LIN {X 0,Y 453.492,Z 301.489,A -85,B 0,C 180,E1 -8435.264,E2 -8435.264} C_VEL
LIN {X 0,Y 453.473,Z 301.492,A -85,B 0,C 180,E1 -8438.414,E2 -8438.414} C_VEL
LIN {X 0,Y 453.514,Z 301.48,A -85,B 0,C 180,E1 -8441.008,E2 -8441.008} C_VEL
LIN {X 0,Y 453.56,Z 301.483,A -85,B 0,C 180,E1 -8443.879,E2 -8443.879} C_VEL
LIN {X 0,Y 453.555,Z 301.485,A -85,B 0,C 180,E1 -8447.47,E2 -8447.47} C_VEL
LIN {X 0,Y 453.584,Z 301.465,A -85,B 0,C 180,E1 -8451.086,E2 -8451.086} C_VEL
LIN {X 0,Y 453.668,Z 301.472,A -85,B 0,C 180,E1 -8453.774,E2 -8453.774} C_VEL
LIN {X 0,Y 453.755,Z 301.46,A -85,B 0,C 180,E1 -8457.336,E2 -8457.336} C_VEL
LIN {X 0,Y 453.812,Z 301.433,A -85,B 0,C 180,E1 -8460,E2 -8460} C_VEL
LIN {X 0,Y 453.735,Z 301.456,A -85,B 0,C 180,E1 -8462.663,E2 -8462.663} C_VEL
LIN {X 0,Y 453.667,Z 301.47,A -85,B 0,C 180,E1 -8466.225,E2 -8466.225} C_VEL
LIN {X 0,Y 453.583,Z 301.473,A -85,B 0,C 180,E1 -8468.913,E2 -8468.913} C_VEL
LIN {X 0,Y 453.553,Z 301.48,A -85,B 0,C 180,E1 -8472.529,E2 -8472.529} C_VEL
LIN {X 0,Y 453.534,Z 301.486,A -85,B 0,C 180,E1 -8476.196,E2 -8476.196} C_VEL
LIN {X 0,Y 453.51,Z 301.48,A -85,B 0,C 180,E1 -8479.04,E2 -8479.04} C_VEL
LIN {X 0,Y 453.466,Z 301.493,A -85,B 0,C 180,E1 -8481.836,E2 -8481.836} C_VEL
LIN {X 0,Y 453.504,Z 301.496,A -85,B 0,C 180,E1 -8484.734,E2 -8484.734} C_VEL
LIN {X 0,Y 453.523,Z 301.478,A -85,B 0,C 180,E1 -8487.96,E2 -8487.96} C_VEL
LIN {X 0,Y 453.474,Z 301.501,A -85,B 0,C 180,E1 -8490.759,E2 -8490.759} C_VEL
LIN {X 0,Y 453.468,Z 301.489,A -85,B 0,C 180,E1 -8493.913,E2 -8493.913} C_VEL
LIN {X 0,Y 453.462,Z 301.499,A -85,B 0,C 180,E1 -8497.188,E2 -8497.188} C_VEL
LIN {X 0,Y 453.522,Z 301.486,A -85,B 0,C 180,E1 -8499.446,E2 -8499.446} C_VEL
LIN {X 0,Y 453.481,Z 301.498,A -85,B 0,C 180,E1 -8502.992,E2 -8502.992} C_VEL
LIN {X 0,Y 453.465,Z 301.49,A -85,B 0,C 180,E1 -8505.78,E2 -8505.78} C_VEL
LIN {X 0,Y 453.507,Z 301.481,A -85,B 0,C 180,E1 -8509.406,E2 -8509.406} C_VEL
LIN {X 0,Y 453.466,Z 301.501,A -85,B 0,C 180,E1 -8512.224,E2 -8512.224} C_VEL
LIN {X 0,Y 453.482,Z 301.478,A -85,B 0,C 180,E1 -8515.223,E2 -8515.223} C_VEL
LIN {X 0,Y 453.461,Z 301.502,A -85,B 0,C 180,E1 -8518.475,E2 -8518.475} C_VEL
LIN {X 0,Y 453.532,Z 301.487,A -85,B 0,C 180,E1 -8522.039,E2 -8522.039} C_VEL
LIN {X 0,Y 453.509,Z 301.493,A -85,B 0,C 180,E1 -8525.266,E2 -8525.266} C_VEL
LIN {X 0,Y 453.475,Z 301.501,A -85,B 0,C 180,E1 -8528.415,E2 -8528.415} C_VEL
LIN {X 0,Y 453.517,Z 301.493,A -85,B 0,C 180,E1 -8531.009,E2 -8531.009} C_VEL
LIN {X 0,Y 453.564,Z 301.49,A -85,B 0,C 180,E1 -8533.88,E2 -8533.88} C_VEL
LIN {X 0,Y 453.559,Z 301.488,A -85,B 0,C 180,E1 -8537.471,E2 -8537.471} C_VEL
LIN {X 0,Y 453.589,Z 301.484,A -85,B 0,C 180,E1 -8541.087,E2 -8541.087} C_VEL
LIN {X 0,Y 453.634,Z 301.478,A -85,B 0,C 180,E1 -8543.101,E2 -8543.101} C_VEL
LIN {X 0,Y 452.949,Z 301.567,A -85,B 0,C 180,E1 -8543.841,E2 -8543.841} C_VEL
LIN {X 0,Y 450.001,Z 301.932,A -85,B 0,C 180,E1 -8545.043,E2 -8545.043} C_VEL
LIN {X 0,Y 447.578,Z 302.236,A -85,B 0,C 180,E1 -8546.012,E2 -8546.012} C_VEL
LIN {X 0,Y 446.643,Z 302.351,A -85,B 0,C 180,E1 -8546.763,E2 -8546.763} C_VEL
LIN {X 0,Y 446.623,Z 302.352,A -85,B 0,C 180,E1 -8547.016,E2 -8547.016} C_VEL
LIN {X 0,Y 446.791,Z 302.334,A -85,B 0,C 180,E1 -8550,E2 -8550} C_VEL
LIN {X 0,Y 446.706,Z 302.342,A -85,B 0,C 180,E1 -8552.705,E2 -8552.705} C_VEL
LIN {X 0,Y 446.644,Z 302.351,A -85,B 0,C 180,E1 -8556.324,E2 -8556.324} C_VEL
LIN {X 0,Y 446.534,Z 302.364,A -85,B 0,C 180,E1 -8559.055,E2 -8559.055} C_VEL
LIN {X 0,Y 446.517,Z 302.365,A -85,B 0,C 180,E1 -8562.73,E2 -8562.73} C_VEL
LIN {X 0,Y 446.492,Z 302.37,A -85,B 0,C 180,E1 -8566.228,E2 -8566.228} C_VEL
LIN {X 0,Y 446.465,Z 302.373,A -85,B 0,C 180,E1 -8569.303,E2 -8569.303} C_VEL
LIN {X 0,Y 446.414,Z 302.379,A -85,B 0,C 180,E1 -8572.199,E2 -8572.199} C_VEL
LIN {X 0,Y 446.453,Z 302.374,A -85,B 0,C 180,E1 -8575.152,E2 -8575.152} C_VEL
LIN {X 0,Y 446.479,Z 302.363,A -85,B 0,C 180,E1 -8578.178,E2 -8578.178} C_VEL
LIN {X 0,Y 446.414,Z 302.379,A -85,B 0,C 180,E1 -8581.775,E2 -8581.775} C_VEL
LIN {X 0,Y 446.423,Z 302.356,A -85,B 0,C 180,E1 -8584.523,E2 -8584.523} C_VEL
LIN {X 0,Y 446.425,Z 302.375,A -85,B 0,C 180,E1 -8588.082,E2 -8588.082} C_VEL
LIN {X 0,Y 446.435,Z 302.358,A -85,B 0,C 180,E1 -8590.92,E2 -8590.92} C_VEL
LIN {X 0,Y 446.414,Z 302.367,A -85,B 0,C 180,E1 -8593.843,E2 -8593.843} C_VEL
LIN {X 0,Y 446.436,Z 302.372,A -85,B 0,C 180,E1 -8596.397,E2 -8596.397} C_VEL
LIN {X 0,Y 446.46,Z 302.367,A -85,B 0,C 180,E1 -8599.805,E2 -8599.805} C_VEL
LIN {X 0,Y 446.424,Z 302.374,A -85,B 0,C 180,E1 -8602.123,E2 -8602.123} C_VEL
LIN {X 0,Y 446.421,Z 302.368,A -85,B 0,C 180,E1 -8605.477,E2 -8605.477} C_VEL
LIN {X 0,Y 446.41,Z 302.377,A -85,B 0,C 180,E1 -8608.7,E2 -8608.7} C_VEL
LIN {X 0,Y 446.475,Z 302.356,A -85,B 0,C 180,E1 -8611.821,E2 -8611.821} C_VEL
LIN {X 0,Y 446.447,Z 302.369,A -85,B 0,C 180,E1 -8614.848,E2 -8614.848} C_VEL
LIN {X 0,Y 446.438,Z 302.369,A -85,B 0,C 180,E1 -8618.245,E2 -8618.245} C_VEL
LIN {X 0,Y 446.447,Z 302.361,A -85,B 0,C 180,E1 -8621.649,E2 -8621.649} C_VEL
LIN {X 0,Y 446.498,Z 302.364,A -85,B 0,C 180,E1 -8624.48,E2 -8624.48} C_VEL
LIN {X 0,Y 446.506,Z 302.359,A -85,B 0,C 180,E1 -8627.384,E2 -8627.384} C_VEL
LIN {X 0,Y 446.528,Z 302.348,A -85,B 0,C 180,E1 -8630.945,E2 -8630.945} C_VEL
LIN {X 0,Y 446.636,Z 302.346,A -85,B 0,C 180,E1 -8633.677,E2 -8633.677} C_VEL
LIN {X 0,Y 446.682,Z 302.335,A -85,B 0,C 180,E1 -8637.295,E2 -8637.295} C_VEL
LIN {X 0,Y 446.783,Z 302.308,A -85,B 0,C 180,E1 -8640.001,E2 -8640.001} C_VEL
LIN {X 0,Y 446.699,Z 302.339,A -85,B 0,C 180,E1 -8642.706,E2 -8642.706} C_VEL
LIN {X 0,Y 446.637,Z 302.348,A -85,B 0,C 180,E1 -8646.324,E2 -8646.324} C_VEL
LIN {X 0,Y 446.53,Z 302.342,A -85,B 0,C 180,E1 -8649.056,E2 -8649.056} C_VEL
LIN {X 0,Y 446.513,Z 302.365,A -85,B 0,C 180,E1 -8652.73,E2 -8652.73} C_VEL
LIN {X 0,Y 446.488,Z 302.365,A -85,B 0,C 180,E1 -8656.229,E2 -8656.229} C_VEL
LIN {X 0,Y 446.462,Z 302.356,A -85,B 0,C 180,E1 -8659.304,E2 -8659.304} C_VEL
LIN {X 0,Y 446.41,Z 302.376,A -85,B 0,C 180,E1 -8662.2,E2 -8662.2} C_VEL
LIN {X 0,Y 446.436,Z 302.364,A -85,B 0,C 180,E1 -8665.154,E2 -8665.154} C_VEL
LIN {X 0,Y 446.479,Z 302.36,A -85,B 0,C 180,E1 -8668.18,E2 -8668.18} C_VEL
LIN {X 0,Y 446.408,Z 302.374,A -85,B 0,C 180,E1 -8671.301,E2 -8671.301} C_VEL
LIN {X 0,Y 446.416,Z 302.37,A -85,B 0,C 180,E1 -8674.525,E2 -8674.525} C_VEL
LIN {X 0,Y 446.408,Z 302.381,A -85,B 0,C 180,E1 -8678.08,E2 -8678.08} C_VEL
LIN {X 0,Y 446.422,Z 302.372,A -85,B 0,C 180,E1 -8680.918,E2 -8680.918} C_VEL
LIN {X 0,Y 446.395,Z 302.38,A -85,B 0,C 180,E1 -8683.847,E2 -8683.847} C_VEL
LIN {X 0,Y 446.396,Z 302.381,A -85,B 0,C 180,E1 -8686.404,E2 -8686.404} C_VEL
LIN {X 0,Y 446.419,Z 302.361,A -85,B 0,C 180,E1 -8689.084,E2 -8689.084} C_VEL
LIN {X 0,Y 446.403,Z 302.382,A -85,B 0,C 180,E1 -8692.122,E2 -8692.122} C_VEL
LIN {X 0,Y 446.427,Z 302.373,A -85,B 0,C 180,E1 -8695.478,E2 -8695.478} C_VEL
LIN {X 0,Y 446.416,Z 302.38,A -85,B 0,C 180,E1 -8698.7,E2 -8698.7} C_VEL
LIN {X 0,Y 446.523,Z 302.561,A -85,B 0,C 180,E1 -8701.813,E2 -8701.813} C_VEL
LIN {X 0,Y 448.386,Z 312.725,A -85,B 0,C 180,E1 -8704.467,E2 -8704.467} C_VEL
LIN {X 0,Y 448.438,Z 317.528,A -85,B 0,C 180,E1 -8705.649,E2 -8705.649} C_VEL
LIN {X 0,Y 447.685,Z 331.236,A -85,B 0,C 180,E1 -8708.835,E2 -8708.835} C_VEL
LIN {X 0,Y 447.04,Z 343.412,A -85,B 0,C 180,E1 -8711.674,E2 -8711.674} C_VEL
LIN {X 0,Y 446.989,Z 345.405,A -85,B 0,C 180,E1 -8712.117,E2 -8712.117} C_VEL
LIN {X 0,Y 447.514,Z 348.844,A -85,B 0,C 180,E1 -8712.245,E2 -8712.245} C_VEL
LIN {X 0,Y 450.815,Z 368.098,A -85,B 0,C 180,E1 -8712.692,E2 -8712.692} C_VEL
LIN {X 0,Y 450.115,Z 450.358,A -85,B 0,C 180,E1 -8714.027,E2 -8714.027} C_VEL
LIN {X 0,Y 449.794,Z 461.123,A -85,B 0,C 180,E1 -8714.306,E2 -8714.306} C_VEL
LIN {X 0,Y 449.474,Z 470.223,A -85,B 0,C 180,E1 -8714.643,E2 -8714.643} C_VEL
LIN {X 0,Y 448.987,Z 480.584,A -85,B 0,C 180,E1 -8715.149,E2 -8715.149} C_VEL
LIN {X 0,Y 448.533,Z 489.719,A -85,B 0,C 180,E1 -8715.713,E2 -8715.713} C_VEL
LIN {X 0,Y 448.044,Z 498.716,A -85,B 0,C 180,E1 -8716.392,E2 -8716.392} C_VEL
LIN {X 0,Y 447.604,Z 507.306,A -85,B 0,C 180,E1 -8717.172,E2 -8717.172} C_VEL
LIN {X 0,Y 447.186,Z 514.844,A -85,B 0,C 180,E1 -8717.981,E2 -8717.981} C_VEL
LIN {X 0,Y 446.7,Z 522.063,A -85,B 0,C 180,E1 -8718.888,E2 -8718.888} C_VEL
LIN {X 0,Y 446.377,Z 528.266,A -85,B 0,C 180,E1 -8719.798,E2 -8719.798} C_VEL
LIN {X 0,Y 446.006,Z 534.803,A -85,B 0,C 180,E1 -8720.934,E2 -8720.934} C_VEL
LIN {X 0,Y 445.838,Z 539.306,A -85,B 0,C 180,E1 -8721.844,E2 -8721.844} C_VEL
LIN {X 0,Y 445.581,Z 544.797,A -85,B 0,C 180,E1 -8723.207,E2 -8723.207} C_VEL
LIN {X 0,Y 445.479,Z 549.118,A -85,B 0,C 180,E1 -8724.569,E2 -8724.569} C_VEL
LIN {X 0,Y 445.414,Z 551.482,A -85,B 0,C 180,E1 -8725.475,E2 -8725.475} C_VEL
LIN {X 0,Y 445.433,Z 554.666,A -85,B 0,C 180,E1 -8727.287,E2 -8727.287} C_VEL
LIN {X 0,Y 445.356,Z 555.721,A -85,B 0,C 180,E1 -8728.191,E2 -8728.191} C_VEL
LIN {X 0,Y 445.339,Z 556.308,A -85,B 0,C 180,E1 -8729.096,E2 -8729.096} C_VEL
LIN {X 0,Y 445.339,Z 556.308,A -85,B 0,C 180,E1 -8730.904,E2 -8730.904} C_VEL
LIN {X 0,Y 445.356,Z 555.721,A -85,B 0,C 180,E1 -8731.809,E2 -8731.809} C_VEL
LIN {X 0,Y 445.433,Z 554.666,A -85,B 0,C 180,E1 -8732.713,E2 -8732.713} C_VEL
LIN {X 0,Y 445.414,Z 551.482,A -85,B 0,C 180,E1 -8734.525,E2 -8734.525} C_VEL
LIN {X 0,Y 445.471,Z 547.36,A -85,B 0,C 180,E1 -8736.044,E2 -8736.044} C_VEL
LIN {X 0,Y 445.637,Z 543.135,A -85,B 0,C 180,E1 -8737.248,E2 -8737.248} C_VEL
LIN {X 0,Y 445.897,Z 537.114,A -85,B 0,C 180,E1 -8738.611,E2 -8738.611} C_VEL
LIN {X 0,Y 446.217,Z 531.018,A -85,B 0,C 180,E1 -8739.748,E2 -8739.748} C_VEL
LIN {X 0,Y 446.506,Z 525.317,A -85,B 0,C 180,E1 -8740.658,E2 -8740.658} C_VEL
LIN {X 0,Y 447.064,Z 516.763,A -85,B 0,C 180,E1 -8741.792,E2 -8741.792} C_VEL
LIN {X 0,Y 447.541,Z 508.582,A -85,B 0,C 180,E1 -8742.7,E2 -8742.7} C_VEL
LIN {X 0,Y 447.964,Z 500.142,A -85,B 0,C 180,E1 -8743.489,E2 -8743.489} C_VEL
LIN {X 0,Y 448.474,Z 491.352,A -85,B 0,C 180,E1 -8744.173,E2 -8744.173} C_VEL
LIN {X 0,Y 448.961,Z 481.592,A -85,B 0,C 180,E1 -8744.794,E2 -8744.794} C_VEL
LIN {X 0,Y 449.367,Z 472.798,A -85,B 0,C 180,E1 -8745.244,E2 -8745.244} C_VEL
LIN {X 0,Y 449.75,Z 462.871,A -85,B 0,C 180,E1 -8745.637,E2 -8745.637} C_VEL
LIN {X 0,Y 450.049,Z 453.021,A -85,B 0,C 180,E1 -8745.917,E2 -8745.917} C_VEL
LIN {X 0,Y 450.317,Z 427.887,A -85,B 0,C 180,E1 -8746.353,E2 -8746.353} C_VEL
LIN {X 0,Y 450.703,Z 367.244,A -85,B 0,C 180,E1 -8747.326,E2 -8747.326} C_VEL
LIN {X 0,Y 447.009,Z 345.81,A -85,B 0,C 180,E1 -8747.844,E2 -8747.844} C_VEL
LIN {X 0,Y 447.009,Z 344.423,A -85,B 0,C 180,E1 -8748.076,E2 -8748.076} C_VEL
LIN {X 0,Y 447.714,Z 331.421,A -85,B 0,C 180,E1 -8751.164,E2 -8751.164} C_VEL
LIN {X 0,Y 448.576,Z 316.323,A -85,B 0,C 180,E1 -8754.672,E2 -8754.672} C_VEL
LIN {X 0,Y 448.193,Z 311.699,A -85,B 0,C 180,E1 -8755.794,E2 -8755.794} C_VEL
LIN {X 0,Y 446.51,Z 302.392,A -85,B 0,C 180,E1 -8758.259,E2 -8758.259} C_VEL
LIN {X 0,Y 446.419,Z 302.377,A -85,B 0,C 180,E1 -8761.774,E2 -8761.774} C_VEL
LIN {X 0,Y 446.427,Z 302.374,A -85,B 0,C 180,E1 -8764.522,E2 -8764.522} C_VEL
LIN {X 0,Y 446.409,Z 302.38,A -85,B 0,C 180,E1 -8768.078,E2 -8768.078} C_VEL
LIN {X 0,Y 446.416,Z 302.364,A -85,B 0,C 180,E1 -8771.391,E2 -8771.391} C_VEL
LIN {X 0,Y 446.447,Z 302.37,A -85,B 0,C 180,E1 -8775.103,E2 -8775.103} C_VEL
LIN {X 0,Y 446.424,Z 302.372,A -85,B 0,C 180,E1 -8778.608,E2 -8778.608} C_VEL
LIN {X 0,Y 446.433,Z 302.368,A -85,B 0,C 180,E1 -8780.971,E2 -8780.971} C_VEL
LIN {X 0,Y 446.412,Z 302.371,A -85,B 0,C 180,E1 -8784.373,E2 -8784.373} C_VEL
LIN {X 0,Y 446.41,Z 302.374,A -85,B 0,C 180,E1 -8787.637,E2 -8787.637} C_VEL
LIN {X 0,Y 446.442,Z 302.369,A -85,B 0,C 180,E1 -8790.79,E2 -8790.79} C_VEL
LIN {X 0,Y 446.471,Z 302.36,A -85,B 0,C 180,E1 -8793.848,E2 -8793.848} C_VEL
LIN {X 0,Y 446.418,Z 302.373,A -85,B 0,C 180,E1 -8796.822,E2 -8796.822} C_VEL
LIN {X 0,Y 446.437,Z 302.364,A -85,B 0,C 180,E1 -8799.736,E2 -8799.736} C_VEL
LIN {X 0,Y 446.455,Z 302.357,A -85,B 0,C 180,E1 -8802.596,E2 -8802.596} C_VEL
LIN {X 0,Y 446.464,Z 302.373,A -85,B 0,C 180,E1 -8805.412,E2 -8805.412} C_VEL
LIN {X 0,Y 446.51,Z 302.355,A -85,B 0,C 180,E1 -8808.192,E2 -8808.192} C_VEL
LIN {X 0,Y 446.591,Z 302.345,A -85,B 0,C 180,E1 -8811.857,E2 -8811.857} C_VEL
LIN {X 0,Y 446.636,Z 302.346,A -85,B 0,C 180,E1 -8814.582,E2 -8814.582} C_VEL
LIN {X 0,Y 446.699,Z 302.339,A -85,B 0,C 180,E1 -8817.294,E2 -8817.294} C_VEL
LIN {X 0,Y 446.783,Z 302.308,A -85,B 0,C 180,E1 -8819.999,E2 -8819.999} C_VEL
LIN {X 0,Y 446.683,Z 302.335,A -85,B 0,C 180,E1 -8822.705,E2 -8822.705} C_VEL
LIN {X 0,Y 446.636,Z 302.346,A -85,B 0,C 180,E1 -8826.323,E2 -8826.323} C_VEL
LIN {X 0,Y 446.528,Z 302.348,A -85,B 0,C 180,E1 -8829.055,E2 -8829.055} C_VEL
LIN {X 0,Y 446.514,Z 302.359,A -85,B 0,C 180,E1 -8832.729,E2 -8832.729} C_VEL
LIN {X 0,Y 446.486,Z 302.364,A -85,B 0,C 180,E1 -8836.228,E2 -8836.228} C_VEL
LIN {X 0,Y 446.459,Z 302.357,A -85,B 0,C 180,E1 -8839.303,E2 -8839.303} C_VEL
LIN {X 0,Y 446.408,Z 302.373,A -85,B 0,C 180,E1 -8842.2,E2 -8842.2} C_VEL
LIN {X 0,Y 446.447,Z 302.369,A -85,B 0,C 180,E1 -8845.152,E2 -8845.152} C_VEL
LIN {X 0,Y 446.475,Z 302.356,A -85,B 0,C 180,E1 -8848.179,E2 -8848.179} C_VEL
LIN {X 0,Y 446.41,Z 302.377,A -85,B 0,C 180,E1 -8851.3,E2 -8851.3} C_VEL
LIN {X 0,Y 446.421,Z 302.368,A -85,B 0,C 180,E1 -8854.523,E2 -8854.523} C_VEL
LIN {X 0,Y 446.428,Z 302.375,A -85,B 0,C 180,E1 -8858.083,E2 -8858.083} C_VEL
LIN {X 0,Y 446.436,Z 302.369,A -85,B 0,C 180,E1 -8860.921,E2 -8860.921} C_VEL
LIN {X 0,Y 446.434,Z 302.372,A -85,B 0,C 180,E1 -8863.841,E2 -8863.841} C_VEL
LIN {X 0,Y 446.412,Z 302.362,A -85,B 0,C 180,E1 -8866.401,E2 -8866.401} C_VEL
LIN {X 0,Y 446.458,Z 302.36,A -85,B 0,C 180,E1 -8869.805,E2 -8869.805} C_VEL
LIN {X 0,Y 446.421,Z 302.377,A -85,B 0,C 180,E1 -8872.124,E2 -8872.124} C_VEL
LIN {X 0,Y 446.423,Z 302.356,A -85,B 0,C 180,E1 -8875.477,E2 -8875.477} C_VEL
LIN {X 0,Y 446.41,Z 302.377,A -85,B 0,C 180,E1 -8878.7,E2 -8878.7} C_VEL
LIN {X 0,Y 446.479,Z 302.363,A -85,B 0,C 180,E1 -8881.822,E2 -8881.822} C_VEL
LIN {X 0,Y 446.453,Z 302.374,A -85,B 0,C 180,E1 -8884.848,E2 -8884.848} C_VEL
LIN {X 0,Y 446.443,Z 302.377,A -85,B 0,C 180,E1 -8888.245,E2 -8888.245} C_VEL
LIN {X 0,Y 446.453,Z 302.374,A -85,B 0,C 180,E1 -8891.649,E2 -8891.649} C_VEL
LIN {X 0,Y 446.503,Z 302.369,A -85,B 0,C 180,E1 -8894.48,E2 -8894.48} C_VEL
LIN {X 0,Y 446.514,Z 302.369,A -85,B 0,C 180,E1 -8898.193,E2 -8898.193} C_VEL
LIN {X 0,Y 446.596,Z 302.358,A -85,B 0,C 180,E1 -8901.858,E2 -8901.858} C_VEL
LIN {X 0,Y 446.643,Z 302.351,A -85,B 0,C 180,E1 -8904.583,E2 -8904.583} C_VEL
LIN {X 0,Y 446.623,Z 302.352,A -85,B 0,C 180,E1 -8907.016,E2 -8907.016} C_VEL
LIN {X 0,Y 446.106,Z 302.419,A -85,B 0,C 180,E1 -8907.769,E2 -8907.769} C_VEL
LIN {X 0,Y 443.288,Z 302.771,A -85,B 0,C 180,E1 -8908.992,E2 -8908.992} C_VEL
LIN {X 0,Y 440.801,Z 303.081,A -85,B 0,C 180,E1 -8909.979,E2 -8909.979} C_VEL
LIN {X 0,Y 439.712,Z 303.214,A -85,B 0,C 180,E1 -8910.742,E2 -8910.742} C_VEL
LIN {X 0,Y 439.618,Z 303.225,A -85,B 0,C 180,E1 -8911.001,E2 -8911.001} C_VEL
LIN {X 0,Y 439.653,Z 303.221,A -85,B 0,C 180,E1 -8912.749,E2 -8912.749} C_VEL
LIN {X 0,Y 439.615,Z 303.226,A -85,B 0,C 180,E1 -8916.425,E2 -8916.425} C_VEL
LIN {X 0,Y 439.496,Z 303.241,A -85,B 0,C 180,E1 -8919.201,E2 -8919.201} C_VEL
LIN {X 0,Y 439.461,Z 303.244,A -85,B 0,C 180,E1 -8922.937,E2 -8922.937} C_VEL
LIN {X 0,Y 439.443,Z 303.247,A -85,B 0,C 180,E1 -8926.349,E2 -8926.349} C_VEL
LIN {X 0,Y 439.398,Z 303.255,A -85,B 0,C 180,E1 -8929.626,E2 -8929.626} C_VEL
LIN {X 0,Y 439.361,Z 303.256,A -85,B 0,C 180,E1 -8932.575,E2 -8932.575} C_VEL
LIN {X 0,Y 439.401,Z 303.254,A -85,B 0,C 180,E1 -8935.584,E2 -8935.584} C_VEL
LIN {X 0,Y 439.412,Z 303.242,A -85,B 0,C 180,E1 -8938.673,E2 -8938.673} C_VEL
LIN {X 0,Y 439.364,Z 303.255,A -85,B 0,C 180,E1 -8942.03,E2 -8942.03} C_VEL
LIN {X 0,Y 439.389,Z 303.236,A -85,B 0,C 180,E1 -8945.34,E2 -8945.34} C_VEL
LIN {X 0,Y 439.385,Z 303.251,A -85,B 0,C 180,E1 -8948.594,E2 -8948.594} C_VEL
LIN {X 0,Y 439.39,Z 303.228,A -85,B 0,C 180,E1 -8951.258,E2 -8951.258} C_VEL
LIN {X 0,Y 439.398,Z 303.242,A -85,B 0,C 180,E1 -8954.728,E2 -8954.728} C_VEL
LIN {X 0,Y 439.397,Z 303.247,A -85,B 0,C 180,E1 -8957.797,E2 -8957.797} C_VEL
LIN {X 0,Y 439.442,Z 303.239,A -85,B 0,C 180,E1 -8960.23,E2 -8960.23} C_VEL
LIN {X 0,Y 439.368,Z 303.25,A -85,B 0,C 180,E1 -8963.713,E2 -8963.713} C_VEL
LIN {X 0,Y 439.363,Z 303.251,A -85,B 0,C 180,E1 -8967.054,E2 -8967.054} C_VEL
LIN {X 0,Y 439.387,Z 303.248,A -85,B 0,C 180,E1 -8970.275,E2 -8970.275} C_VEL
LIN {X 0,Y 439.419,Z 303.24,A -85,B 0,C 180,E1 -8973.396,E2 -8973.396} C_VEL
LIN {X 0,Y 439.377,Z 303.252,A -85,B 0,C 180,E1 -8976.43,E2 -8976.43} C_VEL
LIN {X 0,Y 439.378,Z 303.241,A -85,B 0,C 180,E1 -8979.397,E2 -8979.397} C_VEL
LIN {X 0,Y 439.421,Z 303.236,A -85,B 0,C 180,E1 -8982.31,E2 -8982.31} C_VEL
LIN {X 0,Y 439.439,Z 303.248,A -85,B 0,C 180,E1 -8985.174,E2 -8985.174} C_VEL
LIN {X 0,Y 439.474,Z 303.232,A -85,B 0,C 180,E1 -8988.002,E2 -8988.002} C_VEL
LIN {X 0,Y 439.538,Z 303.223,A -85,B 0,C 180,E1 -8991.727,E2 -8991.727} C_VEL
LIN {X 0,Y 439.611,Z 303.224,A -85,B 0,C 180,E1 -8994.496,E2 -8994.496} C_VEL
LIN {X 0,Y 439.624,Z 303.212,A -85,B 0,C 180,E1 -8998.168,E2 -8998.168} C_VEL
LIN {X 0,Y 439.753,Z 303.183,A -85,B 0,C 180,E1 -9000.001,E2 -9000.001} C_VEL
LIN {X 0,Y 439.646,Z 303.218,A -85,B 0,C 180,E1 -9002.749,E2 -9002.749} C_VEL
LIN {X 0,Y 439.609,Z 303.225,A -85,B 0,C 180,E1 -9006.426,E2 -9006.426} C_VEL
LIN {X 0,Y 439.492,Z 303.217,A -85,B 0,C 180,E1 -9009.202,E2 -9009.202} C_VEL
LIN {X 0,Y 439.457,Z 303.242,A -85,B 0,C 180,E1 -9012.938,E2 -9012.938} C_VEL
LIN {X 0,Y 439.439,Z 303.242,A -85,B 0,C 180,E1 -9016.349,E2 -9016.349} C_VEL
LIN {X 0,Y 439.395,Z 303.236,A -85,B 0,C 180,E1 -9019.627,E2 -9019.627} C_VEL
LIN {X 0,Y 439.356,Z 303.258,A -85,B 0,C 180,E1 -9022.576,E2 -9022.576} C_VEL
LIN {X 0,Y 439.39,Z 303.242,A -85,B 0,C 180,E1 -9025.586,E2 -9025.586} C_VEL
LIN {X 0,Y 439.411,Z 303.248,A -85,B 0,C 180,E1 -9028.674,E2 -9028.674} C_VEL
LIN {X 0,Y 439.36,Z 303.256,A -85,B 0,C 180,E1 -9032.03,E2 -9032.03} C_VEL
LIN {X 0,Y 439.386,Z 303.245,A -85,B 0,C 180,E1 -9035.341,E2 -9035.341} C_VEL
LIN {X 0,Y 439.366,Z 303.251,A -85,B 0,C 180,E1 -9038.597,E2 -9038.597} C_VEL
LIN {X 0,Y 439.384,Z 303.249,A -85,B 0,C 180,E1 -9041.258,E2 -9041.258} C_VEL
LIN {X 0,Y 439.396,Z 303.249,A -85,B 0,C 180,E1 -9044.731,E2 -9044.731} C_VEL
LIN {X 0,Y 439.381,Z 303.252,A -85,B 0,C 180,E1 -9047.795,E2 -9047.795} C_VEL
LIN {X 0,Y 439.356,Z 303.246,A -85,B 0,C 180,E1 -9050.221,E2 -9050.221} C_VEL
LIN {X 0,Y 439.37,Z 303.249,A -85,B 0,C 180,E1 -9053.713,E2 -9053.713} C_VEL
LIN {X 0,Y 439.372,Z 303.25,A -85,B 0,C 180,E1 -9057.055,E2 -9057.055} C_VEL
LIN {X 0,Y 439.382,Z 303.251,A -85,B 0,C 180,E1 -9060.275,E2 -9060.275} C_VEL
LIN {X 0,Y 439.473,Z 303.463,A -85,B 0,C 180,E1 -9061.589,E2 -9061.589} C_VEL
LIN {X 0,Y 441.198,Z 312.584,A -85,B 0,C 180,E1 -9064.021,E2 -9064.021} C_VEL
LIN {X 0,Y 441.564,Z 316.859,A -85,B 0,C 180,E1 -9065.125,E2 -9065.125} C_VEL
LIN {X 0,Y 440.768,Z 331.067,A -85,B 0,C 180,E1 -9068.486,E2 -9068.486} C_VEL
LIN {X 0,Y 440.064,Z 343.22,A -85,B 0,C 180,E1 -9071.373,E2 -9071.373} C_VEL
LIN {X 0,Y 439.993,Z 345.214,A -85,B 0,C 180,E1 -9071.823,E2 -9071.823} C_VEL
LIN {X 0,Y 440.666,Z 349.188,A -85,B 0,C 180,E1 -9071.968,E2 -9071.968} C_VEL
LIN {X 0,Y 444.03,Z 369.152,A -85,B 0,C 180,E1 -9072.44,E2 -9072.44} C_VEL
LIN {X 0,Y 443.308,Z 450.164,A -85,B 0,C 180,E1 -9073.775,E2 -9073.775} C_VEL
LIN {X 0,Y 442.996,Z 460.054,A -85,B 0,C 180,E1 -9074.029,E2 -9074.029} C_VEL
LIN {X 0,Y 442.605,Z 470.028,A -85,B 0,C 180,E1 -9074.399,E2 -9074.399} C_VEL
LIN {X 0,Y 442.134,Z 480.39,A -85,B 0,C 180,E1 -9074.913,E2 -9074.913} C_VEL
LIN {X 0,Y 441.65,Z 489.525,A -85,B 0,C 180,E1 -9075.486,E2 -9075.486} C_VEL
LIN {X 0,Y 441.127,Z 498.522,A -85,B 0,C 180,E1 -9076.174,E2 -9076.174} C_VEL
LIN {X 0,Y 440.692,Z 506.622,A -85,B 0,C 180,E1 -9076.917,E2 -9076.917} C_VEL
LIN {X 0,Y 440.229,Z 514.65,A -85,B 0,C 180,E1 -9077.788,E2 -9077.788} C_VEL
LIN {X 0,Y 439.717,Z 521.868,A -85,B 0,C 180,E1 -9078.709,E2 -9078.709} C_VEL
LIN {X 0,Y 439.354,Z 528.071,A -85,B 0,C 180,E1 -9079.633,E2 -9079.633} C_VEL
LIN {X 0,Y 438.98,Z 534.609,A -85,B 0,C 180,E1 -9080.788,E2 -9080.788} C_VEL
LIN {X 0,Y 438.768,Z 539.111,A -85,B 0,C 180,E1 -9081.712,E2 -9081.712} C_VEL
LIN {X 0,Y 438.509,Z 544.6,A -85,B 0,C 180,E1 -9083.096,E2 -9083.096} C_VEL
LIN {X 0,Y 438.377,Z 548.923,A -85,B 0,C 180,E1 -9084.48,E2 -9084.48} C_VEL
LIN {X 0,Y 438.343,Z 551.289,A -85,B 0,C 180,E1 -9085.402,E2 -9085.402} C_VEL
LIN {X 0,Y 438.341,Z 554.472,A -85,B 0,C 180,E1 -9087.243,E2 -9087.243} C_VEL
LIN {X 0,Y 438.279,Z 555.527,A -85,B 0,C 180,E1 -9088.162,E2 -9088.162} C_VEL
LIN {X 0,Y 438.252,Z 556.114,A -85,B 0,C 180,E1 -9089.081,E2 -9089.081} C_VEL
LIN {X 0,Y 438.252,Z 556.114,A -85,B 0,C 180,E1 -9090.919,E2 -9090.919} C_VEL
LIN {X 0,Y 438.279,Z 555.527,A -85,B 0,C 180,E1 -9091.838,E2 -9091.838} C_VEL
LIN {X 0,Y 438.341,Z 554.472,A -85,B 0,C 180,E1 -9092.757,E2 -9092.757} C_VEL
LIN {X 0,Y 438.343,Z 551.289,A -85,B 0,C 180,E1 -9094.598,E2 -9094.598} C_VEL
LIN {X 0,Y 438.423,Z 546.486,A -85,B 0,C 180,E1 -9096.344,E2 -9096.344} C_VEL
LIN {X 0,Y 438.667,Z 541.026,A -85,B 0,C 180,E1 -9097.827,E2 -9097.827} C_VEL
LIN {X 0,Y 438.899,Z 535.764,A -85,B 0,C 180,E1 -9098.982,E2 -9098.982} C_VEL
LIN {X 0,Y 439.271,Z 529.447,A -85,B 0,C 180,E1 -9100.136,E2 -9100.136} C_VEL
LIN {X 0,Y 439.591,Z 523.495,A -85,B 0,C 180,E1 -9101.061,E2 -9101.061} C_VEL
LIN {X 0,Y 440.092,Z 516.569,A -85,B 0,C 180,E1 -9101.982,E2 -9101.982} C_VEL
LIN {X 0,Y 440.582,Z 508.388,A -85,B 0,C 180,E1 -9102.904,E2 -9102.904} C_VEL
LIN {X 0,Y 441.017,Z 500.391,A -85,B 0,C 180,E1 -9103.667,E2 -9103.667} C_VEL
LIN {X 0,Y 441.569,Z 491.157,A -85,B 0,C 180,E1 -9104.399,E2 -9104.399} C_VEL
LIN {X 0,Y 442.068,Z 481.397,A -85,B 0,C 180,E1 -9105.03,E2 -9105.03} C_VEL
LIN {X 0,Y 442.556,Z 471.316,A -85,B 0,C 180,E1 -9105.544,E2 -9105.544} C_VEL
LIN {X 0,Y 442.899,Z 461.802,A -85,B 0,C 180,E1 -9105.915,E2 -9105.915} C_VEL
LIN {X 0,Y 443.262,Z 451.495,A -85,B 0,C 180,E1 -9106.197,E2 -9106.197} C_VEL
LIN {X 0,Y 443.93,Z 383.105,A -85,B 0,C 180,E1 -9107.333,E2 -9107.333} C_VEL
LIN {X 0,Y 443.901,Z 367.932,A -85,B 0,C 180,E1 -9107.586,E2 -9107.586} C_VEL
LIN {X 0,Y 440.021,Z 345.599,A -85,B 0,C 180,E1 -9108.139,E2 -9108.139} C_VEL
LIN {X 0,Y 439.997,Z 344.834,A -85,B 0,C 180,E1 -9108.232,E2 -9108.232} C_VEL
LIN {X 0,Y 440.796,Z 331.26,A -85,B 0,C 180,E1 -9111.512,E2 -9111.512} C_VEL
LIN {X 0,Y 441.641,Z 316.975,A -85,B 0,C 180,E1 -9114.897,E2 -9114.897} C_VEL
LIN {X 0,Y 440.988,Z 311.572,A -85,B 0,C 180,E1 -9116.247,E2 -9116.247} C_VEL
LIN {X 0,Y 439.457,Z 303.263,A -85,B 0,C 180,E1 -9118.514,E2 -9118.514} C_VEL
LIN {X 0,Y 439.37,Z 303.252,A -85,B 0,C 180,E1 -9122.029,E2 -9122.029} C_VEL
LIN {X 0,Y 439.392,Z 303.246,A -85,B 0,C 180,E1 -9125.339,E2 -9125.339} C_VEL
LIN {X 0,Y 439.361,Z 303.253,A -85,B 0,C 180,E1 -9128.596,E2 -9128.596} C_VEL
LIN {X 0,Y 439.378,Z 303.239,A -85,B 0,C 180,E1 -9131.255,E2 -9131.255} C_VEL
LIN {X 0,Y 439.396,Z 303.248,A -85,B 0,C 180,E1 -9134.729,E2 -9134.729} C_VEL
LIN {X 0,Y 439.392,Z 303.256,A -85,B 0,C 180,E1 -9137.795,E2 -9137.795} C_VEL
LIN {X 0,Y 439.39,Z 303.247,A -85,B 0,C 180,E1 -9140.223,E2 -9140.223} C_VEL
LIN {X 0,Y 439.368,Z 303.256,A -85,B 0,C 180,E1 -9143.712,E2 -9143.712} C_VEL
LIN {X 0,Y 439.364,Z 303.245,A -85,B 0,C 180,E1 -9147.053,E2 -9147.053} C_VEL
LIN {X 0,Y 439.376,Z 303.25,A -85,B 0,C 180,E1 -9150.273,E2 -9150.273} C_VEL
LIN {X 0,Y 439.421,Z 303.235,A -85,B 0,C 180,E1 -9153.395,E2 -9153.395} C_VEL
LIN {X 0,Y 439.376,Z 303.25,A -85,B 0,C 180,E1 -9156.428,E2 -9156.428} C_VEL
LIN {X 0,Y 439.381,Z 303.247,A -85,B 0,C 180,E1 -9159.396,E2 -9159.396} C_VEL
LIN {X 0,Y 439.423,Z 303.232,A -85,B 0,C 180,E1 -9162.309,E2 -9162.309} C_VEL
LIN {X 0,Y 439.441,Z 303.244,A -85,B 0,C 180,E1 -9165.173,E2 -9165.173} C_VEL
LIN {X 0,Y 439.476,Z 303.232,A -85,B 0,C 180,E1 -9168.001,E2 -9168.001} C_VEL
LIN {X 0,Y 439.539,Z 303.222,A -85,B 0,C 180,E1 -9171.726,E2 -9171.726} C_VEL
LIN {X 0,Y 439.611,Z 303.221,A -85,B 0,C 180,E1 -9174.495,E2 -9174.495} C_VEL
LIN {X 0,Y 439.627,Z 303.212,A -85,B 0,C 180,E1 -9178.167,E2 -9178.167} C_VEL
LIN {X 0,Y 439.753,Z 303.183,A -85,B 0,C 180,E1 -9179.999,E2 -9179.999} C_VEL
LIN {X 0,Y 439.632,Z 303.213,A -85,B 0,C 180,E1 -9182.748,E2 -9182.748} C_VEL
LIN {X 0,Y 439.608,Z 303.222,A -85,B 0,C 180,E1 -9186.425,E2 -9186.425} C_VEL
LIN {X 0,Y 439.49,Z 303.222,A -85,B 0,C 180,E1 -9189.201,E2 -9189.201} C_VEL
LIN {X 0,Y 439.459,Z 303.24,A -85,B 0,C 180,E1 -9192.937,E2 -9192.937} C_VEL
LIN {X 0,Y 439.437,Z 303.243,A -85,B 0,C 180,E1 -9196.348,E2 -9196.348} C_VEL
LIN {X 0,Y 439.392,Z 303.237,A -85,B 0,C 180,E1 -9199.626,E2 -9199.626} C_VEL
LIN {X 0,Y 439.355,Z 303.255,A -85,B 0,C 180,E1 -9202.575,E2 -9202.575} C_VEL
LIN {X 0,Y 439.395,Z 303.243,A -85,B 0,C 180,E1 -9205.585,E2 -9205.585} C_VEL
LIN {X 0,Y 439.415,Z 303.24,A -85,B 0,C 180,E1 -9208.673,E2 -9208.673} C_VEL
LIN {X 0,Y 439.365,Z 303.253,A -85,B 0,C 180,E1 -9211.86,E2 -9211.86} C_VEL
LIN {X 0,Y 439.392,Z 303.246,A -85,B 0,C 180,E1 -9215.156,E2 -9215.156} C_VEL
LIN {X 0,Y 439.389,Z 303.256,A -85,B 0,C 180,E1 -9218.594,E2 -9218.594} C_VEL
LIN {X 0,Y 439.392,Z 303.246,A -85,B 0,C 180,E1 -9221.259,E2 -9221.259} C_VEL
LIN {X 0,Y 439.4,Z 303.247,A -85,B 0,C 180,E1 -9224.729,E2 -9224.729} C_VEL
LIN {X 0,Y 439.39,Z 303.223,A -85,B 0,C 180,E1 -9227.796,E2 -9227.796} C_VEL
LIN {X 0,Y 439.438,Z 303.237,A -85,B 0,C 180,E1 -9230.23,E2 -9230.23} C_VEL
LIN {X 0,Y 439.37,Z 303.25,A -85,B 0,C 180,E1 -9233.713,E2 -9233.713} C_VEL
LIN {X 0,Y 439.367,Z 303.254,A -85,B 0,C 180,E1 -9237.054,E2 -9237.054} C_VEL
LIN {X 0,Y 439.376,Z 303.245,A -85,B 0,C 180,E1 -9240.274,E2 -9240.274} C_VEL
LIN {X 0,Y 439.425,Z 303.247,A -85,B 0,C 180,E1 -9243.397,E2 -9243.397} C_VEL
LIN {X 0,Y 439.382,Z 303.257,A -85,B 0,C 180,E1 -9246.43,E2 -9246.43} C_VEL
LIN {X 0,Y 439.383,Z 303.253,A -85,B 0,C 180,E1 -9249.397,E2 -9249.397} C_VEL
LIN {X 0,Y 439.427,Z 303.251,A -85,B 0,C 180,E1 -9252.31,E2 -9252.31} C_VEL
LIN {X 0,Y 439.443,Z 303.246,A -85,B 0,C 180,E1 -9255.174,E2 -9255.174} C_VEL
LIN {X 0,Y 439.48,Z 303.244,A -85,B 0,C 180,E1 -9258.001,E2 -9258.001} C_VEL
LIN {X 0,Y 439.544,Z 303.236,A -85,B 0,C 180,E1 -9261.726,E2 -9261.726} C_VEL
LIN {X 0,Y 439.618,Z 303.227,A -85,B 0,C 180,E1 -9264.496,E2 -9264.496} C_VEL
LIN {X 0,Y 439.632,Z 303.225,A -85,B 0,C 180,E1 -9268.168,E2 -9268.168} C_VEL
LIN {X 0,Y 439.761,Z 303.21,A -85,B 0,C 180,E1 -9270,E2 -9270} C_VEL
LIN {X 0,Y 439.618,Z 303.225,A -85,B 0,C 180,E1 -9271.001,E2 -9271.001} C_VEL
LIN {X 0,Y 438.903,Z 303.316,A -85,B 0,C 180,E1 -9271.765,E2 -9271.765} C_VEL
LIN {X 0,Y 435.924,Z 303.685,A -85,B 0,C 180,E1 -9273.004,E2 -9273.004} C_VEL
LIN {X 0,Y 433.473,Z 303.993,A -85,B 0,C 180,E1 -9274.004,E2 -9274.004} C_VEL
LIN {X 0,Y 432.501,Z 304.112,A -85,B 0,C 180,E1 -9274.779,E2 -9274.779} C_VEL
LIN {X 0,Y 432.464,Z 304.116,A -85,B 0,C 180,E1 -9275.041,E2 -9275.041} C_VEL
LIN {X 0,Y 432.582,Z 304.103,A -85,B 0,C 180,E1 -9277.679,E2 -9277.679} C_VEL
LIN {X 0,Y 432.389,Z 304.127,A -85,B 0,C 180,E1 -9281.247,E2 -9281.247} C_VEL
LIN {X 0,Y 432.369,Z 304.13,A -85,B 0,C 180,E1 -9284.112,E2 -9284.112} C_VEL
LIN {X 0,Y 432.393,Z 304.125,A -85,B 0,C 180,E1 -9287.011,E2 -9287.011} C_VEL
LIN {X 0,Y 432.334,Z 304.134,A -85,B 0,C 180,E1 -9289.96,E2 -9289.96} C_VEL
LIN {X 0,Y 432.315,Z 304.134,A -85,B 0,C 180,E1 -9292.964,E2 -9292.964} C_VEL
LIN {X 0,Y 432.36,Z 304.13,A -85,B 0,C 180,E1 -9296.032,E2 -9296.032} C_VEL
LIN {X 0,Y 432.337,Z 304.119,A -85,B 0,C 180,E1 -9299.187,E2 -9299.187} C_VEL
LIN {X 0,Y 432.317,Z 304.131,A -85,B 0,C 180,E1 -9302.443,E2 -9302.443} C_VEL
LIN {X 0,Y 432.339,Z 304.117,A -85,B 0,C 180,E1 -9305.632,E2 -9305.632} C_VEL
LIN {X 0,Y 432.347,Z 304.128,A -85,B 0,C 180,E1 -9308.717,E2 -9308.717} C_VEL
LIN {X 0,Y 432.358,Z 304.098,A -85,B 0,C 180,E1 -9311.793,E2 -9311.793} C_VEL
LIN {X 0,Y 432.37,Z 304.128,A -85,B 0,C 180,E1 -9315.658,E2 -9315.658} C_VEL
LIN {X 0,Y 432.361,Z 304.121,A -85,B 0,C 180,E1 -9318.392,E2 -9318.392} C_VEL
LIN {X 0,Y 432.343,Z 304.13,A -85,B 0,C 180,E1 -9321.851,E2 -9321.851} C_VEL
LIN {X 0,Y 432.332,Z 304.122,A -85,B 0,C 180,E1 -9325.323,E2 -9325.323} C_VEL
LIN {X 0,Y 432.315,Z 304.133,A -85,B 0,C 180,E1 -9328.654,E2 -9328.654} C_VEL
LIN {X 0,Y 432.371,Z 304.116,A -85,B 0,C 180,E1 -9331.369,E2 -9331.369} C_VEL
LIN {X 0,Y 432.354,Z 304.12,A -85,B 0,C 180,E1 -9333.968,E2 -9333.968} C_VEL
LIN {X 0,Y 432.309,Z 304.138,A -85,B 0,C 180,E1 -9337.036,E2 -9337.036} C_VEL
LIN {X 0,Y 432.377,Z 304.11,A -85,B 0,C 180,E1 -9340.515,E2 -9340.515} C_VEL
LIN {X 0,Y 432.421,Z 304.116,A -85,B 0,C 180,E1 -9343.961,E2 -9343.961} C_VEL
LIN {X 0,Y 432.45,Z 304.107,A -85,B 0,C 180,E1 -9347.804,E2 -9347.804} C_VEL
LIN {X 0,Y 432.482,Z 304.102,A -85,B 0,C 180,E1 -9351.591,E2 -9351.591} C_VEL
LIN {X 0,Y 432.587,Z 304.098,A -85,B 0,C 180,E1 -9354.407,E2 -9354.407} C_VEL
LIN {X 0,Y 432.594,Z 304.088,A -85,B 0,C 180,E1 -9358.139,E2 -9358.139} C_VEL
LIN {X 0,Y 432.723,Z 304.057,A -85,B 0,C 180,E1 -9360.001,E2 -9360.001} C_VEL
LIN {X 0,Y 432.596,Z 304.097,A -85,B 0,C 180,E1 -9362.794,E2 -9362.794} C_VEL
LIN {X 0,Y 432.563,Z 304.101,A -85,B 0,C 180,E1 -9366.531,E2 -9366.531} C_VEL
LIN {X 0,Y 432.435,Z 304.094,A -85,B 0,C 180,E1 -9369.354,E2 -9369.354} C_VEL
LIN {X 0,Y 432.423,Z 304.12,A -85,B 0,C 180,E1 -9372.804,E2 -9372.804} C_VEL
LIN {X 0,Y 432.405,Z 304.115,A -85,B 0,C 180,E1 -9376.48,E2 -9376.48} C_VEL
LIN {X 0,Y 432.331,Z 304.117,A -85,B 0,C 180,E1 -9379.961,E2 -9379.961} C_VEL
LIN {X 0,Y 432.31,Z 304.132,A -85,B 0,C 180,E1 -9382.965,E2 -9382.965} C_VEL
LIN {X 0,Y 432.354,Z 304.119,A -85,B 0,C 180,E1 -9386.034,E2 -9386.034} C_VEL
LIN {X 0,Y 432.337,Z 304.127,A -85,B 0,C 180,E1 -9389.188,E2 -9389.188} C_VEL
LIN {X 0,Y 432.315,Z 304.128,A -85,B 0,C 180,E1 -9392.444,E2 -9392.444} C_VEL
LIN {X 0,Y 432.332,Z 304.126,A -85,B 0,C 180,E1 -9395.819,E2 -9395.819} C_VEL
LIN {X 0,Y 432.318,Z 304.125,A -85,B 0,C 180,E1 -9399.347,E2 -9399.347} C_VEL
LIN {X 0,Y 432.329,Z 304.13,A -85,B 0,C 180,E1 -9401.798,E2 -9401.798} C_VEL
LIN {X 0,Y 432.33,Z 304.129,A -85,B 0,C 180,E1 -9404.348,E2 -9404.348} C_VEL
LIN {X 0,Y 432.314,Z 304.131,A -85,B 0,C 180,E1 -9407.017,E2 -9407.017} C_VEL
LIN {X 0,Y 432.311,Z 304.119,A -85,B 0,C 180,E1 -9409.825,E2 -9409.825} C_VEL
LIN {X 0,Y 432.303,Z 304.131,A -85,B 0,C 180,E1 -9413.023,E2 -9413.023} C_VEL
LIN {X 0,Y 432.358,Z 304.132,A -85,B 0,C 180,E1 -9415.997,E2 -9415.997} C_VEL
LIN {X 0,Y 432.347,Z 304.13,A -85,B 0,C 180,E1 -9419.491,E2 -9419.491} C_VEL
LIN {X 0,Y 432.45,Z 304.348,A -85,B 0,C 180,E1 -9421.353,E2 -9421.353} C_VEL
LIN {X 0,Y 434.297,Z 314.393,A -85,B 0,C 180,E1 -9424.093,E2 -9424.093} C_VEL
LIN {X 0,Y 434.577,Z 318.467,A -85,B 0,C 180,E1 -9425.136,E2 -9425.136} C_VEL
LIN {X 0,Y 433.801,Z 331.932,A -85,B 0,C 180,E1 -9428.373,E2 -9428.373} C_VEL
LIN {X 0,Y 433.036,Z 343.982,A -85,B 0,C 180,E1 -9431.305,E2 -9431.305} C_VEL
LIN {X 0,Y 433.037,Z 345.305,A -85,B 0,C 180,E1 -9431.551,E2 -9431.551} C_VEL
LIN {X 0,Y 437.154,Z 368.958,A -85,B 0,C 180,E1 -9432.154,E2 -9432.154} C_VEL
LIN {X 0,Y 436.54,Z 448.642,A -85,B 0,C 180,E1 -9433.486,E2 -9433.486} C_VEL
LIN {X 0,Y 436.177,Z 459.861,A -85,B 0,C 180,E1 -9433.773,E2 -9433.773} C_VEL
LIN {X 0,Y 435.78,Z 469.834,A -85,B 0,C 180,E1 -9434.148,E2 -9434.148} C_VEL
LIN {X 0,Y 435.287,Z 480.197,A -85,B 0,C 180,E1 -9434.67,E2 -9434.67} C_VEL
LIN {X 0,Y 434.761,Z 489.33,A -85,B 0,C 180,E1 -9435.25,E2 -9435.25} C_VEL
LIN {X 0,Y 434.212,Z 498.327,A -85,B 0,C 180,E1 -9435.949,E2 -9435.949} C_VEL
LIN {X 0,Y 433.72,Z 506.849,A -85,B 0,C 180,E1 -9436.747,E2 -9436.747} C_VEL
LIN {X 0,Y 433.274,Z 514.455,A -85,B 0,C 180,E1 -9437.589,E2 -9437.589} C_VEL
LIN {X 0,Y 432.745,Z 521.674,A -85,B 0,C 180,E1 -9438.525,E2 -9438.525} C_VEL
LIN {X 0,Y 432.334,Z 527.876,A -85,B 0,C 180,E1 -9439.463,E2 -9439.463} C_VEL
LIN {X 0,Y 431.944,Z 534.414,A -85,B 0,C 180,E1 -9440.636,E2 -9440.636} C_VEL
LIN {X 0,Y 431.698,Z 538.915,A -85,B 0,C 180,E1 -9441.575,E2 -9441.575} C_VEL
LIN {X 0,Y 431.43,Z 544.406,A -85,B 0,C 180,E1 -9442.983,E2 -9442.983} C_VEL
LIN {X 0,Y 431.279,Z 548.729,A -85,B 0,C 180,E1 -9444.389,E2 -9444.389} C_VEL
LIN {X 0,Y 431.272,Z 551.095,A -85,B 0,C 180,E1 -9445.326,E2 -9445.326} C_VEL
LIN {X 0,Y 431.236,Z 554.278,A -85,B 0,C 180,E1 -9447.198,E2 -9447.198} C_VEL
LIN {X 0,Y 431.203,Z 555.334,A -85,B 0,C 180,E1 -9448.132,E2 -9448.132} C_VEL
LIN {X 0,Y 431.169,Z 555.921,A -85,B 0,C 180,E1 -9449.066,E2 -9449.066} C_VEL
LIN {X 0,Y 431.169,Z 555.921,A -85,B 0,C 180,E1 -9450.934,E2 -9450.934} C_VEL
LIN {X 0,Y 431.203,Z 555.334,A -85,B 0,C 180,E1 -9451.868,E2 -9451.868} C_VEL
LIN {X 0,Y 431.188,Z 552.891,A -85,B 0,C 180,E1 -9453.738,E2 -9453.738} C_VEL
LIN {X 0,Y 431.295,Z 549.946,A -85,B 0,C 180,E1 -9455.142,E2 -9455.142} C_VEL
LIN {X 0,Y 431.378,Z 545.959,A -85,B 0,C 180,E1 -9456.548,E2 -9456.548} C_VEL
LIN {X 0,Y 431.594,Z 540.831,A -85,B 0,C 180,E1 -9457.956,E2 -9457.956} C_VEL
LIN {X 0,Y 431.849,Z 535.569,A -85,B 0,C 180,E1 -9459.13,E2 -9459.13} C_VEL
LIN {X 0,Y 432.236,Z 529.252,A -85,B 0,C 180,E1 -9460.303,E2 -9460.303} C_VEL
LIN {X 0,Y 432.608,Z 523.3,A -85,B 0,C 180,E1 -9461.241,E2 -9461.241} C_VEL
LIN {X 0,Y 433.133,Z 516.374,A -85,B 0,C 180,E1 -9462.177,E2 -9462.177} C_VEL
LIN {X 0,Y 433.625,Z 508.193,A -85,B 0,C 180,E1 -9463.115,E2 -9463.115} C_VEL
LIN {X 0,Y 434.122,Z 499.499,A -85,B 0,C 180,E1 -9463.95,E2 -9463.95} C_VEL
LIN {X 0,Y 434.678,Z 490.963,A -85,B 0,C 180,E1 -9464.633,E2 -9464.633} C_VEL
LIN {X 0,Y 435.211,Z 481.203,A -85,B 0,C 180,E1 -9465.273,E2 -9465.273} C_VEL
LIN {X 0,Y 435.708,Z 471.122,A -85,B 0,C 180,E1 -9465.795,E2 -9465.795} C_VEL
LIN {X 0,Y 436.095,Z 461.609,A -85,B 0,C 180,E1 -9466.17,E2 -9466.17} C_VEL
LIN {X 0,Y 436.439,Z 451.301,A -85,B 0,C 180,E1 -9466.458,E2 -9466.458} C_VEL
LIN {X 0,Y 437.042,Z 394.732,A -85,B 0,C 180,E1 -9467.415,E2 -9467.415} C_VEL
LIN {X 0,Y 437.221,Z 369.4,A -85,B 0,C 180,E1 -9467.835,E2 -9467.835} C_VEL
LIN {X 0,Y 433.077,Z 345.725,A -85,B 0,C 180,E1 -9468.423,E2 -9468.423} C_VEL
LIN {X 0,Y 433.01,Z 344.468,A -85,B 0,C 180,E1 -9468.574,E2 -9468.574} C_VEL
LIN {X 0,Y 433.803,Z 332.128,A -85,B 0,C 180,E1 -9471.627,E2 -9471.627} C_VEL
LIN {X 0,Y 434.702,Z 317.641,A -85,B 0,C 180,E1 -9475.125,E2 -9475.125} C_VEL
LIN {X 0,Y 433.436,Z 309.403,A -85,B 0,C 180,E1 -9477.261,E2 -9477.261} C_VEL
LIN {X 0,Y 432.406,Z 304.145,A -85,B 0,C 180,E1 -9478.744,E2 -9478.744} C_VEL
LIN {X 0,Y 432.325,Z 304.128,A -85,B 0,C 180,E1 -9482.292,E2 -9482.292} C_VEL
LIN {X 0,Y 432.338,Z 304.128,A -85,B 0,C 180,E1 -9484.676,E2 -9484.676} C_VEL
LIN {X 0,Y 432.328,Z 304.133,A -85,B 0,C 180,E1 -9488.15,E2 -9488.15} C_VEL
LIN {X 0,Y 432.322,Z 304.121,A -85,B 0,C 180,E1 -9491.6,E2 -9491.6} C_VEL
LIN {X 0,Y 432.331,Z 304.13,A -85,B 0,C 180,E1 -9494.346,E2 -9494.346} C_VEL
LIN {X 0,Y 432.316,Z 304.13,A -85,B 0,C 180,E1 -9497.015,E2 -9497.015} C_VEL
LIN {X 0,Y 432.329,Z 304.126,A -85,B 0,C 180,E1 -9499.82,E2 -9499.82} C_VEL
LIN {X 0,Y 432.301,Z 304.133,A -85,B 0,C 180,E1 -9503.021,E2 -9503.021} C_VEL
LIN {X 0,Y 432.327,Z 304.122,A -85,B 0,C 180,E1 -9506.001,E2 -9506.001} C_VEL
LIN {X 0,Y 432.341,Z 304.133,A -85,B 0,C 180,E1 -9509.489,E2 -9509.489} C_VEL
LIN {X 0,Y 432.384,Z 304.111,A -85,B 0,C 180,E1 -9512.927,E2 -9512.927} C_VEL
LIN {X 0,Y 432.36,Z 304.126,A -85,B 0,C 180,E1 -9516.022,E2 -9516.022} C_VEL
LIN {X 0,Y 432.343,Z 304.126,A -85,B 0,C 180,E1 -9519.045,E2 -9519.045} C_VEL
LIN {X 0,Y 432.37,Z 304.112,A -85,B 0,C 180,E1 -9522.01,E2 -9522.01} C_VEL
LIN {X 0,Y 432.388,Z 304.12,A -85,B 0,C 180,E1 -9524.926,E2 -9524.926} C_VEL
LIN {X 0,Y 432.451,Z 304.108,A -85,B 0,C 180,E1 -9527.803,E2 -9527.803} C_VEL
LIN {X 0,Y 432.483,Z 304.098,A -85,B 0,C 180,E1 -9531.59,E2 -9531.59} C_VEL
LIN {X 0,Y 432.588,Z 304.095,A -85,B 0,C 180,E1 -9534.406,E2 -9534.406} C_VEL
LIN {X 0,Y 432.597,Z 304.088,A -85,B 0,C 180,E1 -9538.137,E2 -9538.137} C_VEL
LIN {X 0,Y 432.723,Z 304.057,A -85,B 0,C 180,E1 -9539.999,E2 -9539.999} C_VEL
LIN {X 0,Y 432.584,Z 304.091,A -85,B 0,C 180,E1 -9542.793,E2 -9542.793} C_VEL
LIN {X 0,Y 432.563,Z 304.1,A -85,B 0,C 180,E1 -9546.53,E2 -9546.53} C_VEL
LIN {X 0,Y 432.433,Z 304.098,A -85,B 0,C 180,E1 -9549.353,E2 -9549.353} C_VEL
LIN {X 0,Y 432.422,Z 304.115,A -85,B 0,C 180,E1 -9552.804,E2 -9552.804} C_VEL
LIN {X 0,Y 432.402,Z 304.12,A -85,B 0,C 180,E1 -9556.479,E2 -9556.479} C_VEL
LIN {X 0,Y 432.328,Z 304.116,A -85,B 0,C 180,E1 -9559.96,E2 -9559.96} C_VEL
LIN {X 0,Y 432.309,Z 304.138,A -85,B 0,C 180,E1 -9562.964,E2 -9562.964} C_VEL
LIN {X 0,Y 432.354,Z 304.12,A -85,B 0,C 180,E1 -9566.032,E2 -9566.032} C_VEL
LIN {X 0,Y 432.343,Z 304.129,A -85,B 0,C 180,E1 -9569.187,E2 -9569.187} C_VEL
LIN {X 0,Y 432.316,Z 304.133,A -85,B 0,C 180,E1 -9572.293,E2 -9572.293} C_VEL
LIN {X 0,Y 432.332,Z 304.122,A -85,B 0,C 180,E1 -9574.677,E2 -9574.677} C_VEL
LIN {X 0,Y 432.343,Z 304.13,A -85,B 0,C 180,E1 -9578.149,E2 -9578.149} C_VEL
LIN {X 0,Y 432.361,Z 304.121,A -85,B 0,C 180,E1 -9581.608,E2 -9581.608} C_VEL
LIN {X 0,Y 432.37,Z 304.128,A -85,B 0,C 180,E1 -9584.342,E2 -9584.342} C_VEL
LIN {X 0,Y 432.358,Z 304.098,A -85,B 0,C 180,E1 -9588.207,E2 -9588.207} C_VEL
LIN {X 0,Y 432.347,Z 304.128,A -85,B 0,C 180,E1 -9591.283,E2 -9591.283} C_VEL
LIN {X 0,Y 432.339,Z 304.117,A -85,B 0,C 180,E1 -9594.368,E2 -9594.368} C_VEL
LIN {X 0,Y 432.317,Z 304.131,A -85,B 0,C 180,E1 -9597.557,E2 -9597.557} C_VEL
LIN {X 0,Y 432.337,Z 304.119,A -85,B 0,C 180,E1 -9600.813,E2 -9600.813} C_VEL
LIN {X 0,Y 432.36,Z 304.13,A -85,B 0,C 180,E1 -9603.968,E2 -9603.968} C_VEL
LIN {X 0,Y 432.315,Z 304.134,A -85,B 0,C 180,E1 -9607.036,E2 -9607.036} C_VEL
LIN {X 0,Y 432.382,Z 304.128,A -85,B 0,C 180,E1 -9610.515,E2 -9610.515} C_VEL
LIN {X 0,Y 432.426,Z 304.123,A -85,B 0,C 180,E1 -9613.961,E2 -9613.961} C_VEL
LIN {X 0,Y 432.455,Z 304.119,A -85,B 0,C 180,E1 -9617.804,E2 -9617.804} C_VEL
LIN {X 0,Y 432.488,Z 304.115,A -85,B 0,C 180,E1 -9621.59,E2 -9621.59} C_VEL
LIN {X 0,Y 432.595,Z 304.102,A -85,B 0,C 180,E1 -9624.406,E2 -9624.406} C_VEL
LIN {X 0,Y 432.602,Z 304.101,A -85,B 0,C 180,E1 -9628.138,E2 -9628.138} C_VEL
LIN {X 0,Y 432.73,Z 304.086,A -85,B 0,C 180,E1 -9630,E2 -9630} C_VEL
LIN {X 0,Y 432.602,Z 304.099,A -85,B 0,C 180,E1 -9632.793,E2 -9632.793} C_VEL
LIN {X 0,Y 432.464,Z 304.116,A -85,B 0,C 180,E1 -9635.041,E2 -9635.041} C_VEL
LIN {X 0,Y 431.905,Z 304.188,A -85,B 0,C 180,E1 -9635.82,E2 -9635.82} C_VEL
LIN {X 0,Y 429.057,Z 304.542,A -85,B 0,C 180,E1 -9637.085,E2 -9637.085} C_VEL
LIN {X 0,Y 426.571,Z 304.852,A -85,B 0,C 180,E1 -9638.106,E2 -9638.106} C_VEL
LIN {X 0,Y 425.489,Z 304.986,A -85,B 0,C 180,E1 -9638.896,E2 -9638.896} C_VEL
LIN {X 0,Y 425.399,Z 304.997,A -85,B 0,C 180,E1 -9639.163,E2 -9639.163} C_VEL
LIN {X 0,Y 425.389,Z 304.997,A -85,B 0,C 180,E1 -9642.904,E2 -9642.904} C_VEL
LIN {X 0,Y 425.357,Z 305.001,A -85,B 0,C 180,E1 -9646.605,E2 -9646.605} C_VEL
LIN {X 0,Y 425.324,Z 305.008,A -85,B 0,C 180,E1 -9649.635,E2 -9649.635} C_VEL
LIN {X 0,Y 425.302,Z 305.01,A -85,B 0,C 180,E1 -9653.365,E2 -9653.365} C_VEL
LIN {X 0,Y 425.343,Z 305.002,A -85,B 0,C 180,E1 -9656.844,E2 -9656.844} C_VEL
LIN {X 0,Y 425.285,Z 304.999,A -85,B 0,C 180,E1 -9659.719,E2 -9659.719} C_VEL
LIN {X 0,Y 425.276,Z 305.007,A -85,B 0,C 180,E1 -9663.048,E2 -9663.048} C_VEL
LIN {X 0,Y 425.278,Z 305.001,A -85,B 0,C 180,E1 -9665.929,E2 -9665.929} C_VEL
LIN {X 0,Y 425.301,Z 305.008,A -85,B 0,C 180,E1 -9669.045,E2 -9669.045} C_VEL
LIN {X 0,Y 425.308,Z 304.975,A -85,B 0,C 180,E1 -9671.962,E2 -9671.962} C_VEL
LIN {X 0,Y 425.307,Z 305.003,A -85,B 0,C 180,E1 -9675.279,E2 -9675.279} C_VEL
LIN {X 0,Y 425.298,Z 305.001,A -85,B 0,C 180,E1 -9678.625,E2 -9678.625} C_VEL
LIN {X 0,Y 425.315,Z 305.004,A -85,B 0,C 180,E1 -9681.104,E2 -9681.104} C_VEL
LIN {X 0,Y 425.291,Z 305.002,A -85,B 0,C 180,E1 -9684.664,E2 -9684.664} C_VEL
LIN {X 0,Y 425.257,Z 305.01,A -85,B 0,C 180,E1 -9688.073,E2 -9688.073} C_VEL
LIN {X 0,Y 425.328,Z 304.993,A -85,B 0,C 180,E1 -9691.368,E2 -9691.368} C_VEL
LIN {X 0,Y 425.285,Z 305.001,A -85,B 0,C 180,E1 -9694.555,E2 -9694.555} C_VEL
LIN {X 0,Y 425.278,Z 305.006,A -85,B 0,C 180,E1 -9697.661,E2 -9697.661} C_VEL
LIN {X 0,Y 425.352,Z 304.984,A -85,B 0,C 180,E1 -9700.704,E2 -9700.704} C_VEL
LIN {X 0,Y 425.378,Z 304.994,A -85,B 0,C 180,E1 -9703.688,E2 -9703.688} C_VEL
LIN {X 0,Y 425.384,Z 304.992,A -85,B 0,C 180,E1 -9707.096,E2 -9707.096} C_VEL
LIN {X 0,Y 425.392,Z 304.973,A -85,B 0,C 180,E1 -9710.491,E2 -9710.491} C_VEL
LIN {X 0,Y 425.52,Z 304.978,A -85,B 0,C 180,E1 -9713.362,E2 -9713.362} C_VEL
LIN {X 0,Y 425.36,Z 304.998,A -85,B 0,C 180,E1 -9715.262,E2 -9715.262} C_VEL
LIN {X 0,Y 425.564,Z 304.963,A -85,B 0,C 180,E1 -9718.108,E2 -9718.108} C_VEL
LIN {X 0,Y 425.693,Z 304.932,A -85,B 0,C 180,E1 -9720.001,E2 -9720.001} C_VEL
LIN {X 0,Y 425.547,Z 304.975,A -85,B 0,C 180,E1 -9722.84,E2 -9722.84} C_VEL
LIN {X 0,Y 425.521,Z 304.976,A -85,B 0,C 180,E1 -9726.64,E2 -9726.64} C_VEL
LIN {X 0,Y 425.393,Z 304.97,A -85,B 0,C 180,E1 -9729.51,E2 -9729.51} C_VEL
LIN {X 0,Y 425.385,Z 304.996,A -85,B 0,C 180,E1 -9732.904,E2 -9732.904} C_VEL
LIN {X 0,Y 425.354,Z 304.991,A -85,B 0,C 180,E1 -9736.606,E2 -9736.606} C_VEL
LIN {X 0,Y 425.321,Z 304.988,A -85,B 0,C 180,E1 -9739.636,E2 -9739.636} C_VEL
LIN {X 0,Y 425.281,Z 305.009,A -85,B 0,C 180,E1 -9742.34,E2 -9742.34} C_VEL
LIN {X 0,Y 425.284,Z 304.998,A -85,B 0,C 180,E1 -9745.447,E2 -9745.447} C_VEL
LIN {X 0,Y 425.342,Z 304.987,A -85,B 0,C 180,E1 -9747.559,E2 -9747.559} C_VEL
LIN {X 0,Y 425.282,Z 305.009,A -85,B 0,C 180,E1 -9750.817,E2 -9750.817} C_VEL
LIN {X 0,Y 425.286,Z 304.999,A -85,B 0,C 180,E1 -9754.285,E2 -9754.285} C_VEL
LIN {X 0,Y 425.273,Z 305.01,A -85,B 0,C 180,E1 -9757.695,E2 -9757.695} C_VEL
LIN {X 0,Y 425.275,Z 305.007,A -85,B 0,C 180,E1 -9760.521,E2 -9760.521} C_VEL
LIN {X 0,Y 425.254,Z 305.01,A -85,B 0,C 180,E1 -9763.352,E2 -9763.352} C_VEL
LIN {X 0,Y 425.253,Z 305.012,A -85,B 0,C 180,E1 -9766.65,E2 -9766.65} C_VEL
LIN {X 0,Y 425.263,Z 304.996,A -85,B 0,C 180,E1 -9769.871,E2 -9769.871} C_VEL
LIN {X 0,Y 425.274,Z 305.009,A -85,B 0,C 180,E1 -9772.49,E2 -9772.49} C_VEL
LIN {X 0,Y 425.306,Z 305.008,A -85,B 0,C 180,E1 -9775.818,E2 -9775.818} C_VEL
LIN {X 0,Y 425.291,Z 305.011,A -85,B 0,C 180,E1 -9779.24,E2 -9779.24} C_VEL
LIN {X 0,Y 425.382,Z 305.187,A -85,B 0,C 180,E1 -9781.087,E2 -9781.087} C_VEL
LIN {X 0,Y 427.08,Z 314.254,A -85,B 0,C 180,E1 -9783.621,E2 -9783.621} C_VEL
LIN {X 0,Y 427.652,Z 319.332,A -85,B 0,C 180,E1 -9784.966,E2 -9784.966} C_VEL
LIN {X 0,Y 426.808,Z 332.797,A -85,B 0,C 180,E1 -9788.254,E2 -9788.254} C_VEL
LIN {X 0,Y 426.052,Z 344.827,A -85,B 0,C 180,E1 -9791.206,E2 -9791.206} C_VEL
LIN {X 0,Y 426.622,Z 348.248,A -85,B 0,C 180,E1 -9791.344,E2 -9791.344} C_VEL
LIN {X 0,Y 430.507,Z 370.558,A -85,B 0,C 180,E1 -9791.9,E2 -9791.9} C_VEL
LIN {X 0,Y 429.723,Z 449.777,A -85,B 0,C 180,E1 -9793.247,E2 -9793.247} C_VEL
LIN {X 0,Y 429.379,Z 459.667,A -85,B 0,C 180,E1 -9793.509,E2 -9793.509} C_VEL
LIN {X 0,Y 428.947,Z 469.64,A -85,B 0,C 180,E1 -9793.889,E2 -9793.889} C_VEL
LIN {X 0,Y 428.44,Z 480.003,A -85,B 0,C 180,E1 -9794.419,E2 -9794.419} C_VEL
LIN {X 0,Y 427.875,Z 489.136,A -85,B 0,C 180,E1 -9795.007,E2 -9795.007} C_VEL
LIN {X 0,Y 427.31,Z 498.133,A -85,B 0,C 180,E1 -9795.718,E2 -9795.718} C_VEL
LIN {X 0,Y 426.769,Z 506.196,A -85,B 0,C 180,E1 -9796.478,E2 -9796.478} C_VEL
LIN {X 0,Y 426.32,Z 514.261,A -85,B 0,C 180,E1 -9797.383,E2 -9797.383} C_VEL
LIN {X 0,Y 425.763,Z 521.479,A -85,B 0,C 180,E1 -9798.334,E2 -9798.334} C_VEL
LIN {X 0,Y 425.303,Z 527.681,A -85,B 0,C 180,E1 -9799.286,E2 -9799.286} C_VEL
LIN {X 0,Y 424.888,Z 534.219,A -85,B 0,C 180,E1 -9800.479,E2 -9800.479} C_VEL
LIN {X 0,Y 424.645,Z 538.721,A -85,B 0,C 180,E1 -9801.434,E2 -9801.434} C_VEL
LIN {X 0,Y 424.358,Z 544.211,A -85,B 0,C 180,E1 -9802.865,E2 -9802.865} C_VEL
LIN {X 0,Y 424.191,Z 548.534,A -85,B 0,C 180,E1 -9804.295,E2 -9804.295} C_VEL
LIN {X 0,Y 424.201,Z 550.901,A -85,B 0,C 180,E1 -9805.248,E2 -9805.248} C_VEL
LIN {X 0,Y 424.132,Z 554.084,A -85,B 0,C 180,E1 -9807.151,E2 -9807.151} C_VEL
LIN {X 0,Y 424.129,Z 555.141,A -85,B 0,C 180,E1 -9808.101,E2 -9808.101} C_VEL
LIN {X 0,Y 424.089,Z 555.727,A -85,B 0,C 180,E1 -9809.05,E2 -9809.05} C_VEL
LIN {X 0,Y 424.089,Z 555.727,A -85,B 0,C 180,E1 -9810.95,E2 -9810.95} C_VEL
LIN {X 0,Y 424.129,Z 555.141,A -85,B 0,C 180,E1 -9811.899,E2 -9811.899} C_VEL
LIN {X 0,Y 424.099,Z 552.697,A -85,B 0,C 180,E1 -9813.801,E2 -9813.801} C_VEL
LIN {X 0,Y 424.207,Z 549.752,A -85,B 0,C 180,E1 -9815.228,E2 -9815.228} C_VEL
LIN {X 0,Y 424.302,Z 545.765,A -85,B 0,C 180,E1 -9816.658,E2 -9816.658} C_VEL
LIN {X 0,Y 424.538,Z 540.636,A -85,B 0,C 180,E1 -9818.089,E2 -9818.089} C_VEL
LIN {X 0,Y 424.814,Z 535.374,A -85,B 0,C 180,E1 -9819.282,E2 -9819.282} C_VEL
LIN {X 0,Y 425.208,Z 529.057,A -85,B 0,C 180,E1 -9820.475,E2 -9820.475} C_VEL
LIN {X 0,Y 425.638,Z 523.106,A -85,B 0,C 180,E1 -9821.428,E2 -9821.428} C_VEL
LIN {X 0,Y 426.18,Z 516.18,A -85,B 0,C 180,E1 -9822.379,E2 -9822.379} C_VEL
LIN {X 0,Y 426.679,Z 507.998,A -85,B 0,C 180,E1 -9823.332,E2 -9823.332} C_VEL
LIN {X 0,Y 427.217,Z 499.222,A -85,B 0,C 180,E1 -9824.188,E2 -9824.188} C_VEL
LIN {X 0,Y 427.792,Z 490.768,A -85,B 0,C 180,E1 -9824.874,E2 -9824.874} C_VEL
LIN {X 0,Y 428.366,Z 481.009,A -85,B 0,C 180,E1 -9825.523,E2 -9825.523} C_VEL
LIN {X 0,Y 428.836,Z 472.216,A -85,B 0,C 180,E1 -9825.993,E2 -9825.993} C_VEL
LIN {X 0,Y 429.258,Z 462.289,A -85,B 0,C 180,E1 -9826.405,E2 -9826.405} C_VEL
LIN {X 0,Y 429.605,Z 452.439,A -85,B 0,C 180,E1 -9826.696,E2 -9826.696} C_VEL
LIN {X 0,Y 429.944,Z 427.628,A -85,B 0,C 180,E1 -9827.145,E2 -9827.145} C_VEL
LIN {X 0,Y 430.417,Z 369.511,A -85,B 0,C 180,E1 -9828.122,E2 -9828.122} C_VEL
LIN {X 0,Y 426.057,Z 345.1,A -85,B 0,C 180,E1 -9828.762,E2 -9828.762} C_VEL
LIN {X 0,Y 426.083,Z 343.789,A -85,B 0,C 180,E1 -9829.011,E2 -9829.011} C_VEL
LIN {X 0,Y 427.053,Z 329.69,A -85,B 0,C 180,E1 -9832.549,E2 -9832.549} C_VEL
LIN {X 0,Y 427.724,Z 318.333,A -85,B 0,C 180,E1 -9835.348,E2 -9835.348} C_VEL
LIN {X 0,Y 426.163,Z 309.256,A -85,B 0,C 180,E1 -9837.766,E2 -9837.766} C_VEL
LIN {X 0,Y 425.345,Z 305.022,A -85,B 0,C 180,E1 -9839.012,E2 -9839.012} C_VEL
LIN {X 0,Y 425.281,Z 305.004,A -85,B 0,C 180,E1 -9842.562,E2 -9842.562} C_VEL
LIN {X 0,Y 425.297,Z 305.001,A -85,B 0,C 180,E1 -9845.335,E2 -9845.335} C_VEL
LIN {X 0,Y 425.279,Z 305.006,A -85,B 0,C 180,E1 -9848.9,E2 -9848.9} C_VEL
LIN {X 0,Y 425.28,Z 305.002,A -85,B 0,C 180,E1 -9851.956,E2 -9851.956} C_VEL
LIN {X 0,Y 425.282,Z 305.007,A -85,B 0,C 180,E1 -9855.282,E2 -9855.282} C_VEL
LIN {X 0,Y 425.27,Z 305.007,A -85,B 0,C 180,E1 -9858.62,E2 -9858.62} C_VEL
LIN {X 0,Y 425.292,Z 305.001,A -85,B 0,C 180,E1 -9861.1,E2 -9861.1} C_VEL
LIN {X 0,Y 425.29,Z 305.001,A -85,B 0,C 180,E1 -9864.663,E2 -9864.663} C_VEL
LIN {X 0,Y 425.257,Z 305.012,A -85,B 0,C 180,E1 -9868.072,E2 -9868.072} C_VEL
LIN {X 0,Y 425.325,Z 305.001,A -85,B 0,C 180,E1 -9871.367,E2 -9871.367} C_VEL
LIN {X 0,Y 425.347,Z 304.987,A -85,B 0,C 180,E1 -9873.504,E2 -9873.504} C_VEL
LIN {X 0,Y 425.277,Z 305.006,A -85,B 0,C 180,E1 -9876.633,E2 -9876.633} C_VEL
LIN {X 0,Y 425.288,Z 304.997,A -85,B 0,C 180,E1 -9879.694,E2 -9879.694} C_VEL
LIN {X 0,Y 425.334,Z 304.987,A -85,B 0,C 180,E1 -9882.697,E2 -9882.697} C_VEL
LIN {X 0,Y 425.341,Z 305.002,A -85,B 0,C 180,E1 -9885.649,E2 -9885.649} C_VEL
LIN {X 0,Y 425.345,Z 304.991,A -85,B 0,C 180,E1 -9888.563,E2 -9888.563} C_VEL
LIN {X 0,Y 425.529,Z 304.966,A -85,B 0,C 180,E1 -9892.407,E2 -9892.407} C_VEL
LIN {X 0,Y 425.545,Z 304.973,A -85,B 0,C 180,E1 -9894.313,E2 -9894.313} C_VEL
LIN {X 0,Y 425.566,Z 304.963,A -85,B 0,C 180,E1 -9898.107,E2 -9898.107} C_VEL
LIN {X 0,Y 425.693,Z 304.932,A -85,B 0,C 180,E1 -9899.999,E2 -9899.999} C_VEL
LIN {X 0,Y 425.538,Z 304.969,A -85,B 0,C 180,E1 -9902.839,E2 -9902.839} C_VEL
LIN {X 0,Y 425.52,Z 304.978,A -85,B 0,C 180,E1 -9906.638,E2 -9906.638} C_VEL
LIN {X 0,Y 425.392,Z 304.973,A -85,B 0,C 180,E1 -9909.509,E2 -9909.509} C_VEL
LIN {X 0,Y 425.384,Z 304.992,A -85,B 0,C 180,E1 -9912.904,E2 -9912.904} C_VEL
LIN {X 0,Y 425.351,Z 304.999,A -85,B 0,C 180,E1 -9916.605,E2 -9916.605} C_VEL
LIN {X 0,Y 425.319,Z 304.989,A -85,B 0,C 180,E1 -9919.635,E2 -9919.635} C_VEL
LIN {X 0,Y 425.297,Z 305.007,A -85,B 0,C 180,E1 -9923.365,E2 -9923.365} C_VEL
LIN {X 0,Y 425.337,Z 304.99,A -85,B 0,C 180,E1 -9926.844,E2 -9926.844} C_VEL
LIN {X 0,Y 425.309,Z 305.002,A -85,B 0,C 180,E1 -9929.717,E2 -9929.717} C_VEL
LIN {X 0,Y 425.273,Z 305.004,A -85,B 0,C 180,E1 -9933.048,E2 -9933.048} C_VEL
LIN {X 0,Y 425.276,Z 305.003,A -85,B 0,C 180,E1 -9935.929,E2 -9935.929} C_VEL
LIN {X 0,Y 425.304,Z 305.003,A -85,B 0,C 180,E1 -9939.046,E2 -9939.046} C_VEL
LIN {X 0,Y 425.321,Z 305.006,A -85,B 0,C 180,E1 -9942.646,E2 -9942.646} C_VEL
LIN {X 0,Y 425.291,Z 304.999,A -85,B 0,C 180,E1 -9945.281,E2 -9945.281} C_VEL
LIN {X 0,Y 425.296,Z 304.98,A -85,B 0,C 180,E1 -9948.625,E2 -9948.625} C_VEL
LIN {X 0,Y 425.311,Z 305.006,A -85,B 0,C 180,E1 -9951.104,E2 -9951.104} C_VEL
LIN {X 0,Y 425.294,Z 304.99,A -85,B 0,C 180,E1 -9954.665,E2 -9954.665} C_VEL
LIN {X 0,Y 425.259,Z 305.013,A -85,B 0,C 180,E1 -9958.073,E2 -9958.073} C_VEL
LIN {X 0,Y 425.325,Z 304.996,A -85,B 0,C 180,E1 -9961.368,E2 -9961.368} C_VEL
LIN {X 0,Y 425.291,Z 305.011,A -85,B 0,C 180,E1 -9964.555,E2 -9964.555} C_VEL
LIN {X 0,Y 425.283,Z 305.011,A -85,B 0,C 180,E1 -9967.662,E2 -9967.662} C_VEL
LIN {X 0,Y 425.357,Z 305.003,A -85,B 0,C 180,E1 -9970.704,E2 -9970.704} C_VEL
LIN {X 0,Y 425.384,Z 304.999,A -85,B 0,C 180,E1 -9973.689,E2 -9973.689} C_VEL
LIN {X 0,Y 425.408,Z 304.996,A -85,B 0,C 180,E1 -9977.598,E2 -9977.598} C_VEL
LIN {X 0,Y 425.439,Z 304.993,A -85,B 0,C 180,E1 -9981.45,E2 -9981.45} C_VEL
LIN {X 0,Y 425.551,Z 304.979,A -85,B 0,C 180,E1 -9984.313,E2 -9984.313} C_VEL
LIN {X 0,Y 425.572,Z 304.976,A -85,B 0,C 180,E1 -9988.107,E2 -9988.107} C_VEL
LIN {X 0,Y 425.7,Z 304.961,A -85,B 0,C 180,E1 -9990,E2 -9990} C_VEL
LIN {X 0,Y 425.554,Z 304.977,A -85,B 0,C 180,E1 -9992.84,E2 -9992.84} C_VEL
LIN {X 0,Y 425.528,Z 304.981,A -85,B 0,C 180,E1 -9996.639,E2 -9996.639} C_VEL
LIN {X 0,Y 425.399,Z 304.997,A -85,B 0,C 180,E1 -9999.163,E2 -9999.163} C_VEL
LIN {X 0,Y 424.727,Z 305.082,A -85,B 0,C 180,E1 -9999.953,E2 -9999.953} C_VEL
LIN {X 0,Y 421.878,Z 305.436,A -85,B 0,C 180,E1 -10001.237,E2 -10001.237} C_VEL
LIN {X 0,Y 419.462,Z 305.737,A -85,B 0,C 180,E1 -10002.273,E2 -10002.273} C_VEL
LIN {X 0,Y 418.411,Z 305.867,A -85,B 0,C 180,E1 -10003.074,E2 -10003.074} C_VEL
LIN {X 0,Y 418.317,Z 305.879,A -85,B 0,C 180,E1 -10003.345,E2 -10003.345} C_VEL
LIN {X 0,Y 418.309,Z 305.879,A -85,B 0,C 180,E1 -10006.735,E2 -10006.735} C_VEL
LIN {X 0,Y 418.266,Z 305.887,A -85,B 0,C 180,E1 -10009.79,E2 -10009.79} C_VEL
LIN {X 0,Y 418.233,Z 305.888,A -85,B 0,C 180,E1 -10012.736,E2 -10012.736} C_VEL
LIN {X 0,Y 418.266,Z 305.886,A -85,B 0,C 180,E1 -10015.904,E2 -10015.904} C_VEL
LIN {X 0,Y 418.259,Z 305.872,A -85,B 0,C 180,E1 -10019.162,E2 -10019.162} C_VEL
LIN {X 0,Y 418.251,Z 305.883,A -85,B 0,C 180,E1 -10022.844,E2 -10022.844} C_VEL
LIN {X 0,Y 418.242,Z 305.882,A -85,B 0,C 180,E1 -10026.238,E2 -10026.238} C_VEL
LIN {X 0,Y 418.254,Z 305.876,A -85,B 0,C 180,E1 -10029.68,E2 -10029.68} C_VEL
LIN {X 0,Y 418.239,Z 305.855,A -85,B 0,C 180,E1 -10032.323,E2 -10032.323} C_VEL
LIN {X 0,Y 418.253,Z 305.879,A -85,B 0,C 180,E1 -10035.112,E2 -10035.112} C_VEL
LIN {X 0,Y 418.282,Z 305.877,A -85,B 0,C 180,E1 -10037.773,E2 -10037.773} C_VEL
LIN {X 0,Y 418.257,Z 305.887,A -85,B 0,C 180,E1 -10041.559,E2 -10041.559} C_VEL
LIN {X 0,Y 418.251,Z 305.876,A -85,B 0,C 180,E1 -10045.159,E2 -10045.159} C_VEL
LIN {X 0,Y 418.236,Z 305.889,A -85,B 0,C 180,E1 -10047.472,E2 -10047.472} C_VEL
LIN {X 0,Y 418.268,Z 305.88,A -85,B 0,C 180,E1 -10050.893,E2 -10050.893} C_VEL
LIN {X 0,Y 418.261,Z 305.875,A -85,B 0,C 180,E1 -10054.096,E2 -10054.096} C_VEL
LIN {X 0,Y 418.228,Z 305.888,A -85,B 0,C 180,E1 -10057.264,E2 -10057.264} C_VEL
LIN {X 0,Y 418.273,Z 305.866,A -85,B 0,C 180,E1 -10060.364,E2 -10060.364} C_VEL
LIN {X 0,Y 418.307,Z 305.877,A -85,B 0,C 180,E1 -10063.405,E2 -10063.405} C_VEL
LIN {X 0,Y 418.337,Z 305.871,A -85,B 0,C 180,E1 -10066.999,E2 -10066.999} C_VEL
LIN {X 0,Y 418.332,Z 305.85,A -85,B 0,C 180,E1 -10070.329,E2 -10070.329} C_VEL
LIN {X 0,Y 418.483,Z 305.856,A -85,B 0,C 180,E1 -10073.249,E2 -10073.249} C_VEL
LIN {X 0,Y 418.33,Z 305.875,A -85,B 0,C 180,E1 -10075.182,E2 -10075.182} C_VEL
LIN {X 0,Y 418.533,Z 305.838,A -85,B 0,C 180,E1 -10078.076,E2 -10078.076} C_VEL
LIN {X 0,Y 418.662,Z 305.807,A -85,B 0,C 180,E1 -10080.001,E2 -10080.001} C_VEL
LIN {X 0,Y 418.501,Z 305.853,A -85,B 0,C 180,E1 -10082.888,E2 -10082.888} C_VEL
LIN {X 0,Y 418.484,Z 305.85,A -85,B 0,C 180,E1 -10086.752,E2 -10086.752} C_VEL
LIN {X 0,Y 418.333,Z 305.849,A -85,B 0,C 180,E1 -10089.672,E2 -10089.672} C_VEL
LIN {X 0,Y 418.338,Z 305.872,A -85,B 0,C 180,E1 -10093.001,E2 -10093.001} C_VEL
LIN {X 0,Y 418.305,Z 305.867,A -85,B 0,C 180,E1 -10096.736,E2 -10096.736} C_VEL
LIN {X 0,Y 418.263,Z 305.867,A -85,B 0,C 180,E1 -10099.791,E2 -10099.791} C_VEL
LIN {X 0,Y 418.224,Z 305.888,A -85,B 0,C 180,E1 -10102.737,E2 -10102.737} C_VEL
LIN {X 0,Y 418.261,Z 305.874,A -85,B 0,C 180,E1 -10105.905,E2 -10105.905} C_VEL
LIN {X 0,Y 418.259,Z 305.88,A -85,B 0,C 180,E1 -10109.163,E2 -10109.163} C_VEL
LIN {X 0,Y 418.245,Z 305.876,A -85,B 0,C 180,E1 -10112.843,E2 -10112.843} C_VEL
LIN {X 0,Y 418.239,Z 305.886,A -85,B 0,C 180,E1 -10116.239,E2 -10116.239} C_VEL
LIN {X 0,Y 418.238,Z 305.88,A -85,B 0,C 180,E1 -10119.684,E2 -10119.684} C_VEL
LIN {X 0,Y 418.226,Z 305.891,A -85,B 0,C 180,E1 -10122.322,E2 -10122.322} C_VEL
LIN {X 0,Y 418.233,Z 305.884,A -85,B 0,C 180,E1 -10125.11,E2 -10125.11} C_VEL
LIN {X 0,Y 418.231,Z 305.885,A -85,B 0,C 180,E1 -10127.767,E2 -10127.767} C_VEL
LIN {X 0,Y 418.236,Z 305.885,A -85,B 0,C 180,E1 -10131.558,E2 -10131.558} C_VEL
LIN {X 0,Y 418.258,Z 305.881,A -85,B 0,C 180,E1 -10135.16,E2 -10135.16} C_VEL
LIN {X 0,Y 418.245,Z 305.88,A -85,B 0,C 180,E1 -10137.473,E2 -10137.473} C_VEL
LIN {X 0,Y 418.277,Z 305.958,A -85,B 0,C 180,E1 -10140.771,E2 -10140.771} C_VEL
LIN {X 0,Y 419.902,Z 314.129,A -85,B 0,C 180,E1 -10143.135,E2 -10143.135} C_VEL
LIN {X 0,Y 420.705,Z 320.611,A -85,B 0,C 180,E1 -10144.893,E2 -10144.893} C_VEL
LIN {X 0,Y 419.746,Z 334.696,A -85,B 0,C 180,E1 -10148.386,E2 -10148.386} C_VEL
LIN {X 0,Y 419.085,Z 344.632,A -85,B 0,C 180,E1 -10150.882,E2 -10150.882} C_VEL
LIN {X 0,Y 419.635,Z 347.973,A -85,B 0,C 180,E1 -10151.02,E2 -10151.02} C_VEL
LIN {X 0,Y 423.656,Z 370.639,A -85,B 0,C 180,E1 -10151.602,E2 -10151.602} C_VEL
LIN {X 0,Y 422.942,Z 449.584,A -85,B 0,C 180,E1 -10152.97,E2 -10152.97} C_VEL
LIN {X 0,Y 422.589,Z 459.474,A -85,B 0,C 180,E1 -10153.236,E2 -10153.236} C_VEL
LIN {X 0,Y 422.12,Z 469.446,A -85,B 0,C 180,E1 -10153.621,E2 -10153.621} C_VEL
LIN {X 0,Y 421.578,Z 479.808,A -85,B 0,C 180,E1 -10154.159,E2 -10154.159} C_VEL
LIN {X 0,Y 420.989,Z 488.941,A -85,B 0,C 180,E1 -10154.756,E2 -10154.756} C_VEL
LIN {X 0,Y 420.401,Z 497.938,A -85,B 0,C 180,E1 -10155.478,E2 -10155.478} C_VEL
LIN {X 0,Y 419.832,Z 506.001,A -85,B 0,C 180,E1 -10156.251,E2 -10156.251} C_VEL
LIN {X 0,Y 419.357,Z 514.066,A -85,B 0,C 180,E1 -10157.17,E2 -10157.17} C_VEL
LIN {X 0,Y 418.768,Z 521.284,A -85,B 0,C 180,E1 -10158.136,E2 -10158.136} C_VEL
LIN {X 0,Y 418.301,Z 527.486,A -85,B 0,C 180,E1 -10159.105,E2 -10159.105} C_VEL
LIN {X 0,Y 417.845,Z 534.023,A -85,B 0,C 180,E1 -10160.317,E2 -10160.317} C_VEL
LIN {X 0,Y 417.579,Z 538.526,A -85,B 0,C 180,E1 -10161.288,E2 -10161.288} C_VEL
LIN {X 0,Y 417.285,Z 544.016,A -85,B 0,C 180,E1 -10162.743,E2 -10162.743} C_VEL
LIN {X 0,Y 417.109,Z 548.34,A -85,B 0,C 180,E1 -10164.198,E2 -10164.198} C_VEL
LIN {X 0,Y 417.108,Z 550.707,A -85,B 0,C 180,E1 -10165.167,E2 -10165.167} C_VEL
LIN {X 0,Y 417.029,Z 553.889,A -85,B 0,C 180,E1 -10167.102,E2 -10167.102} C_VEL
LIN {X 0,Y 417.057,Z 554.947,A -85,B 0,C 180,E1 -10168.069,E2 -10168.069} C_VEL
LIN {X 0,Y 417.011,Z 555.534,A -85,B 0,C 180,E1 -10169.034,E2 -10169.034} C_VEL
LIN {X 0,Y 417.011,Z 555.534,A -85,B 0,C 180,E1 -10170.966,E2 -10170.966} C_VEL
LIN {X 0,Y 417.057,Z 554.947,A -85,B 0,C 180,E1 -10171.931,E2 -10171.931} C_VEL
LIN {X 0,Y 417.015,Z 552.503,A -85,B 0,C 180,E1 -10173.865,E2 -10173.865} C_VEL
LIN {X 0,Y 417.122,Z 549.557,A -85,B 0,C 180,E1 -10175.317,E2 -10175.317} C_VEL
LIN {X 0,Y 417.235,Z 545.57,A -85,B 0,C 180,E1 -10176.771,E2 -10176.771} C_VEL
LIN {X 0,Y 417.475,Z 540.441,A -85,B 0,C 180,E1 -10178.227,E2 -10178.227} C_VEL
LIN {X 0,Y 417.78,Z 535.179,A -85,B 0,C 180,E1 -10179.44,E2 -10179.44} C_VEL
LIN {X 0,Y 418.181,Z 528.862,A -85,B 0,C 180,E1 -10180.653,E2 -10180.653} C_VEL
LIN {X 0,Y 418.645,Z 522.911,A -85,B 0,C 180,E1 -10181.621,E2 -10181.621} C_VEL
LIN {X 0,Y 419.207,Z 515.985,A -85,B 0,C 180,E1 -10182.588,E2 -10182.588} C_VEL
LIN {X 0,Y 419.719,Z 507.802,A -85,B 0,C 180,E1 -10183.557,E2 -10183.557} C_VEL
LIN {X 0,Y 420.303,Z 499.152,A -85,B 0,C 180,E1 -10184.415,E2 -10184.415} C_VEL
LIN {X 0,Y 420.906,Z 490.574,A -85,B 0,C 180,E1 -10185.123,E2 -10185.123} C_VEL
LIN {X 0,Y 421.537,Z 480.816,A -85,B 0,C 180,E1 -10185.781,E2 -10185.781} C_VEL
LIN {X 0,Y 421.987,Z 472.021,A -85,B 0,C 180,E1 -10186.26,E2 -10186.26} C_VEL
LIN {X 0,Y 422.463,Z 462.096,A -85,B 0,C 180,E1 -10186.676,E2 -10186.676} C_VEL
LIN {X 0,Y 422.826,Z 452.245,A -85,B 0,C 180,E1 -10186.972,E2 -10186.972} C_VEL
LIN {X 0,Y 423.154,Z 429.429,A -85,B 0,C 180,E1 -10187.394,E2 -10187.394} C_VEL
LIN {X 0,Y 423.65,Z 370.302,A -85,B 0,C 180,E1 -10188.404,E2 -10188.404} C_VEL
LIN {X 0,Y 419.126,Z 345.193,A -85,B 0,C 180,E1 -10189.066,E2 -10189.066} C_VEL
LIN {X 0,Y 419.089,Z 344.09,A -85,B 0,C 180,E1 -10189.214,E2 -10189.214} C_VEL
LIN {X 0,Y 420.063,Z 330.774,A -85,B 0,C 180,E1 -10192.631,E2 -10192.631} C_VEL
LIN {X 0,Y 420.762,Z 320.821,A -85,B 0,C 180,E1 -10195.118,E2 -10195.118} C_VEL
LIN {X 0,Y 420.106,Z 315.279,A -85,B 0,C 180,E1 -10196.583,E2 -10196.583} C_VEL
LIN {X 0,Y 418.282,Z 305.922,A -85,B 0,C 180,E1 -10199.246,E2 -10199.246} C_VEL
LIN {X 0,Y 418.257,Z 305.88,A -85,B 0,C 180,E1 -10202.843,E2 -10202.843} C_VEL
LIN {X 0,Y 418.242,Z 305.879,A -85,B 0,C 180,E1 -10206.237,E2 -10206.237} C_VEL
LIN {X 0,Y 418.209,Z 305.879,A -85,B 0,C 180,E1 -10209.686,E2 -10209.686} C_VEL
LIN {X 0,Y 418.221,Z 305.888,A -85,B 0,C 180,E1 -10212.319,E2 -10212.319} C_VEL
LIN {X 0,Y 418.233,Z 305.884,A -85,B 0,C 180,E1 -10215.108,E2 -10215.108} C_VEL
LIN {X 0,Y 418.236,Z 305.891,A -85,B 0,C 180,E1 -10217.766,E2 -10217.766} C_VEL
LIN {X 0,Y 418.241,Z 305.879,A -85,B 0,C 180,E1 -10220.62,E2 -10220.62} C_VEL
LIN {X 0,Y 418.237,Z 305.883,A -85,B 0,C 180,E1 -10223.975,E2 -10223.975} C_VEL
LIN {X 0,Y 418.237,Z 305.88,A -85,B 0,C 180,E1 -10227.471,E2 -10227.471} C_VEL
LIN {X 0,Y 418.263,Z 305.88,A -85,B 0,C 180,E1 -10230.895,E2 -10230.895} C_VEL
LIN {X 0,Y 418.261,Z 305.874,A -85,B 0,C 180,E1 -10234.095,E2 -10234.095} C_VEL
LIN {X 0,Y 418.224,Z 305.888,A -85,B 0,C 180,E1 -10237.263,E2 -10237.263} C_VEL
LIN {X 0,Y 418.276,Z 305.865,A -85,B 0,C 180,E1 -10240.363,E2 -10240.363} C_VEL
LIN {X 0,Y 418.309,Z 305.868,A -85,B 0,C 180,E1 -10243.404,E2 -10243.404} C_VEL
LIN {X 0,Y 418.338,Z 305.872,A -85,B 0,C 180,E1 -10246.999,E2 -10246.999} C_VEL
LIN {X 0,Y 418.333,Z 305.849,A -85,B 0,C 180,E1 -10250.328,E2 -10250.328} C_VEL
LIN {X 0,Y 418.484,Z 305.85,A -85,B 0,C 180,E1 -10253.248,E2 -10253.248} C_VEL
LIN {X 0,Y 418.331,Z 305.877,A -85,B 0,C 180,E1 -10255.181,E2 -10255.181} C_VEL
LIN {X 0,Y 418.536,Z 305.839,A -85,B 0,C 180,E1 -10258.075,E2 -10258.075} C_VEL
LIN {X 0,Y 418.662,Z 305.807,A -85,B 0,C 180,E1 -10259.999,E2 -10259.999} C_VEL
LIN {X 0,Y 418.493,Z 305.847,A -85,B 0,C 180,E1 -10262.887,E2 -10262.887} C_VEL
LIN {X 0,Y 418.483,Z 305.856,A -85,B 0,C 180,E1 -10266.751,E2 -10266.751} C_VEL
LIN {X 0,Y 418.332,Z 305.85,A -85,B 0,C 180,E1 -10269.671,E2 -10269.671} C_VEL
LIN {X 0,Y 418.337,Z 305.871,A -85,B 0,C 180,E1 -10273.001,E2 -10273.001} C_VEL
LIN {X 0,Y 418.303,Z 305.877,A -85,B 0,C 180,E1 -10276.735,E2 -10276.735} C_VEL
LIN {X 0,Y 418.261,Z 305.867,A -85,B 0,C 180,E1 -10279.79,E2 -10279.79} C_VEL
LIN {X 0,Y 418.228,Z 305.888,A -85,B 0,C 180,E1 -10282.736,E2 -10282.736} C_VEL
LIN {X 0,Y 418.261,Z 305.875,A -85,B 0,C 180,E1 -10285.904,E2 -10285.904} C_VEL
LIN {X 0,Y 418.266,Z 305.881,A -85,B 0,C 180,E1 -10289.161,E2 -10289.161} C_VEL
LIN {X 0,Y 418.248,Z 305.882,A -85,B 0,C 180,E1 -10292.844,E2 -10292.844} C_VEL
LIN {X 0,Y 418.24,Z 305.881,A -85,B 0,C 180,E1 -10296.239,E2 -10296.239} C_VEL
LIN {X 0,Y 418.257,Z 305.878,A -85,B 0,C 180,E1 -10299.68,E2 -10299.68} C_VEL
LIN {X 0,Y 418.274,Z 305.879,A -85,B 0,C 180,E1 -10302.329,E2 -10302.329} C_VEL
LIN {X 0,Y 418.247,Z 305.878,A -85,B 0,C 180,E1 -10305.112,E2 -10305.112} C_VEL
LIN {X 0,Y 418.25,Z 305.853,A -85,B 0,C 180,E1 -10307.769,E2 -10307.769} C_VEL
LIN {X 0,Y 418.257,Z 305.88,A -85,B 0,C 180,E1 -10310.618,E2 -10310.618} C_VEL
LIN {X 0,Y 418.239,Z 305.879,A -85,B 0,C 180,E1 -10313.976,E2 -10313.976} C_VEL
LIN {X 0,Y 418.251,Z 305.883,A -85,B 0,C 180,E1 -10317.156,E2 -10317.156} C_VEL
LIN {X 0,Y 418.263,Z 305.872,A -85,B 0,C 180,E1 -10320.896,E2 -10320.896} C_VEL
LIN {X 0,Y 418.266,Z 305.886,A -85,B 0,C 180,E1 -10324.096,E2 -10324.096} C_VEL
LIN {X 0,Y 418.233,Z 305.888,A -85,B 0,C 180,E1 -10327.264,E2 -10327.264} C_VEL
LIN {X 0,Y 418.279,Z 305.885,A -85,B 0,C 180,E1 -10330.364,E2 -10330.364} C_VEL
LIN {X 0,Y 418.313,Z 305.879,A -85,B 0,C 180,E1 -10333.405,E2 -10333.405} C_VEL
LIN {X 0,Y 418.342,Z 305.875,A -85,B 0,C 180,E1 -10336.999,E2 -10336.999} C_VEL
LIN {X 0,Y 418.338,Z 305.878,A -85,B 0,C 180,E1 -10340.329,E2 -10340.329} C_VEL
LIN {X 0,Y 418.49,Z 305.858,A -85,B 0,C 180,E1 -10343.249,E2 -10343.249} C_VEL
LIN {X 0,Y 418.337,Z 305.877,A -85,B 0,C 180,E1 -10345.182,E2 -10345.182} C_VEL
LIN {X 0,Y 418.541,Z 305.852,A -85,B 0,C 180,E1 -10348.076,E2 -10348.076} C_VEL
LIN {X 0,Y 418.669,Z 305.837,A -85,B 0,C 180,E1 -10350,E2 -10350} C_VEL
LIN {X 0,Y 418.507,Z 305.855,A -85,B 0,C 180,E1 -10352.888,E2 -10352.888} C_VEL
LIN {X 0,Y 418.49,Z 305.858,A -85,B 0,C 180,E1 -10356.751,E2 -10356.751} C_VEL
LIN {X 0,Y 418.338,Z 305.878,A -85,B 0,C 180,E1 -10359.671,E2 -10359.671} C_VEL
LIN {X 0,Y 418.317,Z 305.879,A -85,B 0,C 180,E1 -10363.345,E2 -10363.345} C_VEL
LIN {X 0,Y 417.625,Z 305.967,A -85,B 0,C 180,E1 -10364.148,E2 -10364.148} C_VEL
LIN {X 0,Y 414.746,Z 306.325,A -85,B 0,C 180,E1 -10365.454,E2 -10365.454} C_VEL
LIN {X 0,Y 412.333,Z 306.624,A -85,B 0,C 180,E1 -10366.508,E2 -10366.508} C_VEL
LIN {X 0,Y 411.312,Z 306.752,A -85,B 0,C 180,E1 -10367.323,E2 -10367.323} C_VEL
LIN {X 0,Y 411.236,Z 306.76,A -85,B 0,C 180,E1 -10367.599,E2 -10367.599} C_VEL
LIN {X 0,Y 411.192,Z 306.766,A -85,B 0,C 180,E1 -10371.034,E2 -10371.034} C_VEL
LIN {X 0,Y 411.222,Z 306.762,A -85,B 0,C 180,E1 -10374.215,E2 -10374.215} C_VEL
LIN {X 0,Y 411.253,Z 306.759,A -85,B 0,C 180,E1 -10377.477,E2 -10377.477} C_VEL
LIN {X 0,Y 411.183,Z 306.762,A -85,B 0,C 180,E1 -10380.847,E2 -10380.847} C_VEL
LIN {X 0,Y 411.199,Z 306.741,A -85,B 0,C 180,E1 -10384.333,E2 -10384.333} C_VEL
LIN {X 0,Y 411.195,Z 306.765,A -85,B 0,C 180,E1 -10387.973,E2 -10387.973} C_VEL
LIN {X 0,Y 411.192,Z 306.736,A -85,B 0,C 180,E1 -10391.234,E2 -10391.234} C_VEL
LIN {X 0,Y 411.18,Z 306.756,A -85,B 0,C 180,E1 -10394.488,E2 -10394.488} C_VEL
LIN {X 0,Y 411.219,Z 306.763,A -85,B 0,C 180,E1 -10397.297,E2 -10397.297} C_VEL
LIN {X 0,Y 411.222,Z 306.756,A -85,B 0,C 180,E1 -10400.777,E2 -10400.777} C_VEL
LIN {X 0,Y 411.191,Z 306.758,A -85,B 0,C 180,E1 -10404.471,E2 -10404.471} C_VEL
LIN {X 0,Y 411.198,Z 306.756,A -85,B 0,C 180,E1 -10406.873,E2 -10406.873} C_VEL
LIN {X 0,Y 411.232,Z 306.757,A -85,B 0,C 180,E1 -10410.642,E2 -10410.642} C_VEL
LIN {X 0,Y 411.228,Z 306.751,A -85,B 0,C 180,E1 -10413.619,E2 -10413.619} C_VEL
LIN {X 0,Y 411.194,Z 306.766,A -85,B 0,C 180,E1 -10416.853,E2 -10416.853} C_VEL
LIN {X 0,Y 411.205,Z 306.746,A -85,B 0,C 180,E1 -10420.051,E2 -10420.051} C_VEL
LIN {X 0,Y 411.254,Z 306.752,A -85,B 0,C 180,E1 -10423.131,E2 -10423.131} C_VEL
LIN {X 0,Y 411.296,Z 306.75,A -85,B 0,C 180,E1 -10426.896,E2 -10426.896} C_VEL
LIN {X 0,Y 411.284,Z 306.727,A -85,B 0,C 180,E1 -10430.162,E2 -10430.162} C_VEL
LIN {X 0,Y 411.446,Z 306.733,A -85,B 0,C 180,E1 -10433.133,E2 -10433.133} C_VEL
LIN {X 0,Y 411.301,Z 306.751,A -85,B 0,C 180,E1 -10435.099,E2 -10435.099} C_VEL
LIN {X 0,Y 411.502,Z 306.714,A -85,B 0,C 180,E1 -10438.043,E2 -10438.043} C_VEL
LIN {X 0,Y 411.632,Z 306.682,A -85,B 0,C 180,E1 -10440.001,E2 -10440.001} C_VEL
LIN {X 0,Y 411.457,Z 306.731,A -85,B 0,C 180,E1 -10442.938,E2 -10442.938} C_VEL
LIN {X 0,Y 411.447,Z 306.725,A -85,B 0,C 180,E1 -10446.868,E2 -10446.868} C_VEL
LIN {X 0,Y 411.285,Z 306.726,A -85,B 0,C 180,E1 -10449.839,E2 -10449.839} C_VEL
LIN {X 0,Y 411.298,Z 306.749,A -85,B 0,C 180,E1 -10453.105,E2 -10453.105} C_VEL
LIN {X 0,Y 411.256,Z 306.743,A -85,B 0,C 180,E1 -10456.87,E2 -10456.87} C_VEL
LIN {X 0,Y 411.224,Z 306.745,A -85,B 0,C 180,E1 -10459.988,E2 -10459.988} C_VEL
LIN {X 0,Y 411.189,Z 306.762,A -85,B 0,C 180,E1 -10463.149,E2 -10463.149} C_VEL
LIN {X 0,Y 411.23,Z 306.744,A -85,B 0,C 180,E1 -10466.382,E2 -10466.382} C_VEL
LIN {X 0,Y 411.195,Z 306.761,A -85,B 0,C 180,E1 -10469.714,E2 -10469.714} C_VEL
LIN {X 0,Y 411.199,Z 306.752,A -85,B 0,C 180,E1 -10473.157,E2 -10473.157} C_VEL
LIN {X 0,Y 411.187,Z 306.767,A -85,B 0,C 180,E1 -10476.553,E2 -10476.553} C_VEL
LIN {X 0,Y 411.203,Z 306.756,A -85,B 0,C 180,E1 -10479.728,E2 -10479.728} C_VEL
LIN {X 0,Y 411.17,Z 306.764,A -85,B 0,C 180,E1 -10483.135,E2 -10483.135} C_VEL
LIN {X 0,Y 411.165,Z 306.768,A -85,B 0,C 180,E1 -10485.882,E2 -10485.882} C_VEL
LIN {X 0,Y 411.155,Z 306.753,A -85,B 0,C 180,E1 -10488.774,E2 -10488.774} C_VEL
LIN {X 0,Y 411.185,Z 306.769,A -85,B 0,C 180,E1 -10492.026,E2 -10492.026} C_VEL
LIN {X 0,Y 411.205,Z 306.763,A -85,B 0,C 180,E1 -10495.667,E2 -10495.667} C_VEL
LIN {X 0,Y 411.19,Z 306.768,A -85,B 0,C 180,E1 -10499.153,E2 -10499.153} C_VEL
LIN {X 0,Y 411.264,Z 306.978,A -85,B 0,C 180,E1 -10500.573,E2 -10500.573} C_VEL
LIN {X 0,Y 413.176,Z 316.887,A -85,B 0,C 180,E1 -10503.481,E2 -10503.481} C_VEL
LIN {X 0,Y 413.726,Z 322.098,A -85,B 0,C 180,E1 -10504.87,E2 -10504.87} C_VEL
LIN {X 0,Y 412.755,Z 335.561,A -85,B 0,C 180,E1 -10508.264,E2 -10508.264} C_VEL
LIN {X 0,Y 412.148,Z 344.437,A -85,B 0,C 180,E1 -10510.547,E2 -10510.547} C_VEL
LIN {X 0,Y 412.703,Z 347.879,A -85,B 0,C 180,E1 -10510.691,E2 -10510.691} C_VEL
LIN {X 0,Y 416.971,Z 371.952,A -85,B 0,C 180,E1 -10511.323,E2 -10511.323} C_VEL
LIN {X 0,Y 416.177,Z 449.39,A -85,B 0,C 180,E1 -10512.685,E2 -10512.685} C_VEL
LIN {X 0,Y 415.783,Z 459.279,A -85,B 0,C 180,E1 -10512.953,E2 -10512.953} C_VEL
LIN {X 0,Y 415.308,Z 469.252,A -85,B 0,C 180,E1 -10513.345,E2 -10513.345} C_VEL
LIN {X 0,Y 414.817,Z 478.607,A -85,B 0,C 180,E1 -10513.83,E2 -10513.83} C_VEL
LIN {X 0,Y 414.121,Z 488.746,A -85,B 0,C 180,E1 -10514.497,E2 -10514.497} C_VEL
LIN {X 0,Y 413.504,Z 497.743,A -85,B 0,C 180,E1 -10515.23,E2 -10515.23} C_VEL
LIN {X 0,Y 412.879,Z 506.335,A -85,B 0,C 180,E1 -10516.073,E2 -10516.073} C_VEL
LIN {X 0,Y 412.404,Z 513.871,A -85,B 0,C 180,E1 -10516.95,E2 -10516.95} C_VEL
LIN {X 0,Y 411.787,Z 521.089,A -85,B 0,C 180,E1 -10517.932,E2 -10517.932} C_VEL
LIN {X 0,Y 411.309,Z 527.292,A -85,B 0,C 180,E1 -10518.917,E2 -10518.917} C_VEL
LIN {X 0,Y 410.823,Z 533.829,A -85,B 0,C 180,E1 -10520.15,E2 -10520.15} C_VEL
LIN {X 0,Y 410.537,Z 538.331,A -85,B 0,C 180,E1 -10521.137,E2 -10521.137} C_VEL
LIN {X 0,Y 410.206,Z 543.822,A -85,B 0,C 180,E1 -10522.617,E2 -10522.617} C_VEL
LIN {X 0,Y 410.014,Z 548.145,A -85,B 0,C 180,E1 -10524.097,E2 -10524.097} C_VEL
LIN {X 0,Y 410.02,Z 550.513,A -85,B 0,C 180,E1 -10525.084,E2 -10525.084} C_VEL
LIN {X 0,Y 409.933,Z 552.309,A -85,B 0,C 180,E1 -10526.068,E2 -10526.068} C_VEL
LIN {X 0,Y 409.967,Z 554.754,A -85,B 0,C 180,E1 -10528.035,E2 -10528.035} C_VEL
LIN {X 0,Y 409.936,Z 555.341,A -85,B 0,C 180,E1 -10529.018,E2 -10529.018} C_VEL
LIN {X 0,Y 409.936,Z 555.341,A -85,B 0,C 180,E1 -10530.982,E2 -10530.982} C_VEL
LIN {X 0,Y 409.967,Z 554.754,A -85,B 0,C 180,E1 -10531.965,E2 -10531.965} C_VEL
LIN {X 0,Y 409.933,Z 552.309,A -85,B 0,C 180,E1 -10533.932,E2 -10533.932} C_VEL
LIN {X 0,Y 410.018,Z 549.362,A -85,B 0,C 180,E1 -10535.409,E2 -10535.409} C_VEL
LIN {X 0,Y 410.168,Z 545.376,A -85,B 0,C 180,E1 -10536.889,E2 -10536.889} C_VEL
LIN {X 0,Y 410.426,Z 540.247,A -85,B 0,C 180,E1 -10538.369,E2 -10538.369} C_VEL
LIN {X 0,Y 410.752,Z 534.985,A -85,B 0,C 180,E1 -10539.603,E2 -10539.603} C_VEL
LIN {X 0,Y 411.165,Z 528.667,A -85,B 0,C 180,E1 -10540.837,E2 -10540.837} C_VEL
LIN {X 0,Y 411.668,Z 522.717,A -85,B 0,C 180,E1 -10541.821,E2 -10541.821} C_VEL
LIN {X 0,Y 412.235,Z 515.79,A -85,B 0,C 180,E1 -10542.805,E2 -10542.805} C_VEL
LIN {X 0,Y 412.795,Z 507.608,A -85,B 0,C 180,E1 -10543.789,E2 -10543.789} C_VEL
LIN {X 0,Y 413.411,Z 499.079,A -85,B 0,C 180,E1 -10544.649,E2 -10544.649} C_VEL
LIN {X 0,Y 414.031,Z 490.379,A -85,B 0,C 180,E1 -10545.38,E2 -10545.38} C_VEL
LIN {X 0,Y 414.674,Z 480.621,A -85,B 0,C 180,E1 -10546.049,E2 -10546.049} C_VEL
LIN {X 0,Y 415.165,Z 471.827,A -85,B 0,C 180,E1 -10546.535,E2 -10546.535} C_VEL
LIN {X 0,Y 415.675,Z 461.902,A -85,B 0,C 180,E1 -10546.957,E2 -10546.957} C_VEL
LIN {X 0,Y 416.05,Z 452.052,A -85,B 0,C 180,E1 -10547.257,E2 -10547.257} C_VEL
LIN {X 0,Y 416.389,Z 429.236,A -85,B 0,C 180,E1 -10547.686,E2 -10547.686} C_VEL
LIN {X 0,Y 416.926,Z 371.248,A -85,B 0,C 180,E1 -10548.692,E2 -10548.692} C_VEL
LIN {X 0,Y 412.167,Z 344.714,A -85,B 0,C 180,E1 -10549.42,E2 -10549.42} C_VEL
LIN {X 0,Y 412.197,Z 343.403,A -85,B 0,C 180,E1 -10549.678,E2 -10549.678} C_VEL
LIN {X 0,Y 413.165,Z 330.612,A -85,B 0,C 180,E1 -10553.031,E2 -10553.031} C_VEL
LIN {X 0,Y 413.768,Z 321.108,A -85,B 0,C 180,E1 -10555.454,E2 -10555.454} C_VEL
LIN {X 0,Y 412.496,Z 313.15,A -85,B 0,C 180,E1 -10557.629,E2 -10557.629} C_VEL
LIN {X 0,Y 411.242,Z 306.849,A -85,B 0,C 180,E1 -10559.485,E2 -10559.485} C_VEL
LIN {X 0,Y 411.206,Z 306.759,A -85,B 0,C 180,E1 -10563.155,E2 -10563.155} C_VEL
LIN {X 0,Y 411.19,Z 306.76,A -85,B 0,C 180,E1 -10566.551,E2 -10566.551} C_VEL
LIN {X 0,Y 411.177,Z 306.754,A -85,B 0,C 180,E1 -10569.721,E2 -10569.721} C_VEL
LIN {X 0,Y 411.168,Z 306.766,A -85,B 0,C 180,E1 -10573.133,E2 -10573.133} C_VEL
LIN {X 0,Y 411.165,Z 306.765,A -85,B 0,C 180,E1 -10575.88,E2 -10575.88} C_VEL
LIN {X 0,Y 411.159,Z 306.765,A -85,B 0,C 180,E1 -10578.771,E2 -10578.771} C_VEL
LIN {X 0,Y 411.187,Z 306.767,A -85,B 0,C 180,E1 -10582.025,E2 -10582.025} C_VEL
LIN {X 0,Y 411.187,Z 306.754,A -85,B 0,C 180,E1 -10585.664,E2 -10585.664} C_VEL
LIN {X 0,Y 411.183,Z 306.765,A -85,B 0,C 180,E1 -10589.151,E2 -10589.151} C_VEL
LIN {X 0,Y 411.253,Z 306.741,A -85,B 0,C 180,E1 -10592.521,E2 -10592.521} C_VEL
LIN {X 0,Y 411.206,Z 306.763,A -85,B 0,C 180,E1 -10595.783,E2 -10595.783} C_VEL
LIN {X 0,Y 411.189,Z 306.76,A -85,B 0,C 180,E1 -10598.965,E2 -10598.965} C_VEL
LIN {X 0,Y 411.245,Z 306.741,A -85,B 0,C 180,E1 -10602.084,E2 -10602.084} C_VEL
LIN {X 0,Y 411.253,Z 306.754,A -85,B 0,C 180,E1 -10605.147,E2 -10605.147} C_VEL
LIN {X 0,Y 411.277,Z 306.743,A -85,B 0,C 180,E1 -10608.167,E2 -10608.167} C_VEL
LIN {X 0,Y 411.432,Z 306.722,A -85,B 0,C 180,E1 -10612.188,E2 -10612.188} C_VEL
LIN {X 0,Y 411.466,Z 306.727,A -85,B 0,C 180,E1 -10614.117,E2 -10614.117} C_VEL
LIN {X 0,Y 411.505,Z 306.715,A -85,B 0,C 180,E1 -10618.042,E2 -10618.042} C_VEL
LIN {X 0,Y 411.632,Z 306.682,A -85,B 0,C 180,E1 -10619.999,E2 -10619.999} C_VEL
LIN {X 0,Y 411.45,Z 306.724,A -85,B 0,C 180,E1 -10622.937,E2 -10622.937} C_VEL
LIN {X 0,Y 411.446,Z 306.733,A -85,B 0,C 180,E1 -10626.867,E2 -10626.867} C_VEL
LIN {X 0,Y 411.284,Z 306.727,A -85,B 0,C 180,E1 -10629.838,E2 -10629.838} C_VEL
LIN {X 0,Y 411.296,Z 306.75,A -85,B 0,C 180,E1 -10633.104,E2 -10633.104} C_VEL
LIN {X 0,Y 411.254,Z 306.752,A -85,B 0,C 180,E1 -10636.869,E2 -10636.869} C_VEL
LIN {X 0,Y 411.221,Z 306.744,A -85,B 0,C 180,E1 -10639.987,E2 -10639.987} C_VEL
LIN {X 0,Y 411.193,Z 306.766,A -85,B 0,C 180,E1 -10643.147,E2 -10643.147} C_VEL
LIN {X 0,Y 411.228,Z 306.751,A -85,B 0,C 180,E1 -10646.381,E2 -10646.381} C_VEL
LIN {X 0,Y 411.202,Z 306.759,A -85,B 0,C 180,E1 -10649.712,E2 -10649.712} C_VEL
LIN {X 0,Y 411.197,Z 306.756,A -85,B 0,C 180,E1 -10653.156,E2 -10653.156} C_VEL
LIN {X 0,Y 411.187,Z 306.763,A -85,B 0,C 180,E1 -10656.553,E2 -10656.553} C_VEL
LIN {X 0,Y 411.219,Z 306.754,A -85,B 0,C 180,E1 -10659.73,E2 -10659.73} C_VEL
LIN {X 0,Y 411.213,Z 306.762,A -85,B 0,C 180,E1 -10663.128,E2 -10663.128} C_VEL
LIN {X 0,Y 411.168,Z 306.758,A -85,B 0,C 180,E1 -10665.88,E2 -10665.88} C_VEL
LIN {X 0,Y 411.192,Z 306.736,A -85,B 0,C 180,E1 -10668.766,E2 -10668.766} C_VEL
LIN {X 0,Y 411.195,Z 306.765,A -85,B 0,C 180,E1 -10672.027,E2 -10672.027} C_VEL
LIN {X 0,Y 411.199,Z 306.741,A -85,B 0,C 180,E1 -10675.667,E2 -10675.667} C_VEL
LIN {X 0,Y 411.183,Z 306.762,A -85,B 0,C 180,E1 -10679.153,E2 -10679.153} C_VEL
LIN {X 0,Y 411.253,Z 306.759,A -85,B 0,C 180,E1 -10682.523,E2 -10682.523} C_VEL
LIN {X 0,Y 411.222,Z 306.762,A -85,B 0,C 180,E1 -10685.785,E2 -10685.785} C_VEL
LIN {X 0,Y 411.192,Z 306.766,A -85,B 0,C 180,E1 -10688.966,E2 -10688.966} C_VEL
LIN {X 0,Y 411.248,Z 306.761,A -85,B 0,C 180,E1 -10692.085,E2 -10692.085} C_VEL
LIN {X 0,Y 411.256,Z 306.759,A -85,B 0,C 180,E1 -10695.148,E2 -10695.148} C_VEL
LIN {X 0,Y 411.28,Z 306.757,A -85,B 0,C 180,E1 -10698.167,E2 -10698.167} C_VEL
LIN {X 0,Y 411.478,Z 306.733,A -85,B 0,C 180,E1 -10702.147,E2 -10702.147} C_VEL
LIN {X 0,Y 411.472,Z 306.733,A -85,B 0,C 180,E1 -10704.118,E2 -10704.118} C_VEL
LIN {X 0,Y 411.51,Z 306.728,A -85,B 0,C 180,E1 -10708.043,E2 -10708.043} C_VEL
LIN {X 0,Y 411.639,Z 306.713,A -85,B 0,C 180,E1 -10710,E2 -10710} C_VEL
LIN {X 0,Y 411.463,Z 306.733,A -85,B 0,C 180,E1 -10712.937,E2 -10712.937} C_VEL
LIN {X 0,Y 411.457,Z 306.734,A -85,B 0,C 180,E1 -10716.867,E2 -10716.867} C_VEL
LIN {X 0,Y 411.289,Z 306.755,A -85,B 0,C 180,E1 -10719.839,E2 -10719.839} C_VEL
LIN {X 0,Y 411.278,Z 306.755,A -85,B 0,C 180,E1 -10723.333,E2 -10723.333} C_VEL
LIN {X 0,Y 411.253,Z 306.759,A -85,B 0,C 180,E1 -10726.888,E2 -10726.888} C_VEL
LIN {X 0,Y 411.236,Z 306.76,A -85,B 0,C 180,E1 -10727.599,E2 -10727.599} C_VEL
LIN {X 0,Y 410.576,Z 306.845,A -85,B 0,C 180,E1 -10728.416,E2 -10728.416} C_VEL
LIN {X 0,Y 407.688,Z 307.206,A -85,B 0,C 180,E1 -10729.745,E2 -10729.745} C_VEL
LIN {X 0,Y 405.243,Z 307.509,A -85,B 0,C 180,E1 -10730.817,E2 -10730.817} C_VEL
LIN {X 0,Y 404.207,Z 307.638,A -85,B 0,C 180,E1 -10731.647,E2 -10731.647} C_VEL
LIN {X 0,Y 404.131,Z 307.644,A -85,B 0,C 180,E1 -10731.928,E2 -10731.928} C_VEL
LIN {X 0,Y 404.211,Z 307.637,A -85,B 0,C 180,E1 -10735.296,E2 -10735.296} C_VEL
LIN {X 0,Y 404.19,Z 307.632,A -85,B 0,C 180,E1 -10737.999,E2 -10737.999} C_VEL
LIN {X 0,Y 404.133,Z 307.647,A -85,B 0,C 180,E1 -10741.558,E2 -10741.558} C_VEL
LIN {X 0,Y 404.179,Z 307.615,A -85,B 0,C 180,E1 -10745.016,E2 -10745.016} C_VEL
LIN {X 0,Y 404.154,Z 307.641,A -85,B 0,C 180,E1 -10748.756,E2 -10748.756} C_VEL
LIN {X 0,Y 404.142,Z 307.609,A -85,B 0,C 180,E1 -10751.604,E2 -10751.604} C_VEL
LIN {X 0,Y 404.149,Z 307.632,A -85,B 0,C 180,E1 -10754.523,E2 -10754.523} C_VEL
LIN {X 0,Y 404.197,Z 307.637,A -85,B 0,C 180,E1 -10757.304,E2 -10757.304} C_VEL
LIN {X 0,Y 404.161,Z 307.635,A -85,B 0,C 180,E1 -10759.955,E2 -10759.955} C_VEL
LIN {X 0,Y 404.132,Z 307.646,A -85,B 0,C 180,E1 -10763.124,E2 -10763.124} C_VEL
LIN {X 0,Y 404.136,Z 307.633,A -85,B 0,C 180,E1 -10766.188,E2 -10766.188} C_VEL
LIN {X 0,Y 404.145,Z 307.64,A -85,B 0,C 180,E1 -10769.716,E2 -10769.716} C_VEL
LIN {X 0,Y 404.186,Z 307.622,A -85,B 0,C 180,E1 -10773.123,E2 -10773.123} C_VEL
LIN {X 0,Y 404.168,Z 307.641,A -85,B 0,C 180,E1 -10775.334,E2 -10775.334} C_VEL
LIN {X 0,Y 404.15,Z 307.639,A -85,B 0,C 180,E1 -10778.582,E2 -10778.582} C_VEL
LIN {X 0,Y 404.2,Z 307.621,A -85,B 0,C 180,E1 -10781.762,E2 -10781.762} C_VEL
LIN {X 0,Y 404.198,Z 307.637,A -85,B 0,C 180,E1 -10784.882,E2 -10784.882} C_VEL
LIN {X 0,Y 404.248,Z 307.619,A -85,B 0,C 180,E1 -10787.959,E2 -10787.959} C_VEL
LIN {X 0,Y 404.396,Z 307.599,A -85,B 0,C 180,E1 -10792.129,E2 -10792.129} C_VEL
LIN {X 0,Y 404.413,Z 307.606,A -85,B 0,C 180,E1 -10794.015,E2 -10794.015} C_VEL
LIN {X 0,Y 404.471,Z 307.589,A -85,B 0,C 180,E1 -10798.009,E2 -10798.009} C_VEL
LIN {X 0,Y 404.601,Z 307.557,A -85,B 0,C 180,E1 -10800.001,E2 -10800.001} C_VEL
LIN {X 0,Y 404.414,Z 307.609,A -85,B 0,C 180,E1 -10802.989,E2 -10802.989} C_VEL
LIN {X 0,Y 404.394,Z 307.602,A -85,B 0,C 180,E1 -10806.988,E2 -10806.988} C_VEL
LIN {X 0,Y 404.251,Z 307.603,A -85,B 0,C 180,E1 -10810.012,E2 -10810.012} C_VEL
LIN {X 0,Y 404.259,Z 307.625,A -85,B 0,C 180,E1 -10813.212,E2 -10813.212} C_VEL
LIN {X 0,Y 404.209,Z 307.619,A -85,B 0,C 180,E1 -10817.008,E2 -10817.008} C_VEL
LIN {X 0,Y 404.157,Z 307.628,A -85,B 0,C 180,E1 -10820.352,E2 -10820.352} C_VEL
LIN {X 0,Y 404.153,Z 307.637,A -85,B 0,C 180,E1 -10823.576,E2 -10823.576} C_VEL
LIN {X 0,Y 404.177,Z 307.628,A -85,B 0,C 180,E1 -10825.767,E2 -10825.767} C_VEL
LIN {X 0,Y 404.189,Z 307.623,A -85,B 0,C 180,E1 -10828.001,E2 -10828.001} C_VEL
LIN {X 0,Y 404.133,Z 307.641,A -85,B 0,C 180,E1 -10831.559,E2 -10831.559} C_VEL
LIN {X 0,Y 404.169,Z 307.632,A -85,B 0,C 180,E1 -10835.018,E2 -10835.018} C_VEL
LIN {X 0,Y 404.144,Z 307.636,A -85,B 0,C 180,E1 -10838.759,E2 -10838.759} C_VEL
LIN {X 0,Y 404.119,Z 307.643,A -85,B 0,C 180,E1 -10841.601,E2 -10841.601} C_VEL
LIN {X 0,Y 404.142,Z 307.639,A -85,B 0,C 180,E1 -10844.523,E2 -10844.523} C_VEL
LIN {X 0,Y 404.13,Z 307.642,A -85,B 0,C 180,E1 -10847.296,E2 -10847.296} C_VEL
LIN {X 0,Y 404.13,Z 307.627,A -85,B 0,C 180,E1 -10849.952,E2 -10849.952} C_VEL
LIN {X 0,Y 404.133,Z 307.641,A -85,B 0,C 180,E1 -10853.126,E2 -10853.126} C_VEL
LIN {X 0,Y 404.145,Z 307.644,A -85,B 0,C 180,E1 -10856.189,E2 -10856.189} C_VEL
LIN {X 0,Y 404.191,Z 307.634,A -85,B 0,C 180,E1 -10860.102,E2 -10860.102} C_VEL
LIN {X 0,Y 404.261,Z 308.057,A -85,B 0,C 180,E1 -10860.371,E2 -10860.371} C_VEL
LIN {X 0,Y 406.167,Z 317.749,A -85,B 0,C 180,E1 -10863.264,E2 -10863.264} C_VEL
LIN {X 0,Y 406.738,Z 324,A -85,B 0,C 180,E1 -10864.955,E2 -10864.955} C_VEL
LIN {X 0,Y 405.781,Z 336.423,A -85,B 0,C 180,E1 -10868.139,E2 -10868.139} C_VEL
LIN {X 0,Y 405.189,Z 344.268,A -85,B 0,C 180,E1 -10870.203,E2 -10870.203} C_VEL
LIN {X 0,Y 405.969,Z 348.669,A -85,B 0,C 180,E1 -10870.376,E2 -10870.376} C_VEL
LIN {X 0,Y 410.206,Z 372.332,A -85,B 0,C 180,E1 -10871.014,E2 -10871.014} C_VEL
LIN {X 0,Y 409.403,Z 449.196,A -85,B 0,C 180,E1 -10872.389,E2 -10872.389} C_VEL
LIN {X 0,Y 408.963,Z 459.96,A -85,B 0,C 180,E1 -10872.692,E2 -10872.692} C_VEL
LIN {X 0,Y 408.508,Z 469.058,A -85,B 0,C 180,E1 -10873.059,E2 -10873.059} C_VEL
LIN {X 0,Y 407.93,Z 479.42,A -85,B 0,C 180,E1 -10873.614,E2 -10873.614} C_VEL
LIN {X 0,Y 407.281,Z 488.552,A -85,B 0,C 180,E1 -10874.23,E2 -10874.23} C_VEL
LIN {X 0,Y 406.612,Z 497.549,A -85,B 0,C 180,E1 -10874.974,E2 -10874.974} C_VEL
LIN {X 0,Y 406.014,Z 505.658,A -85,B 0,C 180,E1 -10875.778,E2 -10875.778} C_VEL
LIN {X 0,Y 405.449,Z 513.676,A -85,B 0,C 180,E1 -10876.722,E2 -10876.722} C_VEL
LIN {X 0,Y 404.823,Z 520.895,A -85,B 0,C 180,E1 -10877.722,E2 -10877.722} C_VEL
LIN {X 0,Y 404.311,Z 527.097,A -85,B 0,C 180,E1 -10878.723,E2 -10878.723} C_VEL
LIN {X 0,Y 403.817,Z 533.635,A -85,B 0,C 180,E1 -10879.977,E2 -10879.977} C_VEL
LIN {X 0,Y 403.493,Z 538.136,A -85,B 0,C 180,E1 -10880.981,E2 -10880.981} C_VEL
LIN {X 0,Y 403.154,Z 543.627,A -85,B 0,C 180,E1 -10882.488,E2 -10882.488} C_VEL
LIN {X 0,Y 402.94,Z 547.951,A -85,B 0,C 180,E1 -10883.993,E2 -10883.993} C_VEL
LIN {X 0,Y 402.932,Z 550.318,A -85,B 0,C 180,E1 -10884.997,E2 -10884.997} C_VEL
LIN {X 0,Y 402.853,Z 552.115,A -85,B 0,C 180,E1 -10885.999,E2 -10885.999} C_VEL
LIN {X 0,Y 402.865,Z 554.56,A -85,B 0,C 180,E1 -10888.001,E2 -10888.001} C_VEL
LIN {X 0,Y 402.863,Z 555.148,A -85,B 0,C 180,E1 -10889,E2 -10889} C_VEL
LIN {X 0,Y 402.863,Z 555.148,A -85,B 0,C 180,E1 -10891,E2 -10891} C_VEL
LIN {X 0,Y 402.865,Z 554.56,A -85,B 0,C 180,E1 -10891.999,E2 -10891.999} C_VEL
LIN {X 0,Y 402.853,Z 552.115,A -85,B 0,C 180,E1 -10894.001,E2 -10894.001} C_VEL
LIN {X 0,Y 402.916,Z 549.168,A -85,B 0,C 180,E1 -10895.505,E2 -10895.505} C_VEL
LIN {X 0,Y 403.082,Z 545.181,A -85,B 0,C 180,E1 -10897.01,E2 -10897.01} C_VEL
LIN {X 0,Y 403.365,Z 540.052,A -85,B 0,C 180,E1 -10898.517,E2 -10898.517} C_VEL
LIN {X 0,Y 403.714,Z 534.79,A -85,B 0,C 180,E1 -10899.772,E2 -10899.772} C_VEL
LIN {X 0,Y 404.16,Z 528.472,A -85,B 0,C 180,E1 -10901.027,E2 -10901.027} C_VEL
LIN {X 0,Y 404.694,Z 522.522,A -85,B 0,C 180,E1 -10902.028,E2 -10902.028} C_VEL
LIN {X 0,Y 405.271,Z 515.595,A -85,B 0,C 180,E1 -10903.028,E2 -10903.028} C_VEL
LIN {X 0,Y 405.855,Z 507.413,A -85,B 0,C 180,E1 -10904.03,E2 -10904.03} C_VEL
LIN {X 0,Y 406.506,Z 499.036,A -85,B 0,C 180,E1 -10904.889,E2 -10904.889} C_VEL
LIN {X 0,Y 407.16,Z 490.184,A -85,B 0,C 180,E1 -10905.646,E2 -10905.646} C_VEL
LIN {X 0,Y 407.841,Z 480.426,A -85,B 0,C 180,E1 -10906.325,E2 -10906.325} C_VEL
LIN {X 0,Y 408.342,Z 471.633,A -85,B 0,C 180,E1 -10906.819,E2 -10906.819} C_VEL
LIN {X 0,Y 408.904,Z 461.709,A -85,B 0,C 180,E1 -10907.246,E2 -10907.246} C_VEL
LIN {X 0,Y 409.266,Z 451.858,A -85,B 0,C 180,E1 -10907.553,E2 -10907.553} C_VEL
LIN {X 0,Y 409.608,Z 430.832,A -85,B 0,C 180,E1 -10907.957,E2 -10907.957} C_VEL
LIN {X 0,Y 410.253,Z 372.479,A -85,B 0,C 180,E1 -10908.982,E2 -10908.982} C_VEL
LIN {X 0,Y 405.384,Z 345.671,A -85,B 0,C 180,E1 -10909.709,E2 -10909.709} C_VEL
LIN {X 0,Y 405.204,Z 344.004,A -85,B 0,C 180,E1 -10909.837,E2 -10909.837} C_VEL
LIN {X 0,Y 406.29,Z 330.082,A -85,B 0,C 180,E1 -10913.537,E2 -10913.537} C_VEL
LIN {X 0,Y 406.804,Z 322.197,A -85,B 0,C 180,E1 -10915.588,E2 -10915.588} C_VEL
LIN {X 0,Y 405.437,Z 313.885,A -85,B 0,C 180,E1 -10917.906,E2 -10917.906} C_VEL
LIN {X 0,Y 404.205,Z 307.672,A -85,B 0,C 180,E1 -10919.802,E2 -10919.802} C_VEL
LIN {X 0,Y 404.171,Z 307.637,A -85,B 0,C 180,E1 -10923.419,E2 -10923.419} C_VEL
LIN {X 0,Y 404.14,Z 307.635,A -85,B 0,C 180,E1 -10926.245,E2 -10926.245} C_VEL
LIN {X 0,Y 404.141,Z 307.64,A -85,B 0,C 180,E1 -10928.757,E2 -10928.757} C_VEL
LIN {X 0,Y 404.115,Z 307.632,A -85,B 0,C 180,E1 -10931.598,E2 -10931.598} C_VEL
LIN {X 0,Y 404.142,Z 307.64,A -85,B 0,C 180,E1 -10934.521,E2 -10934.521} C_VEL
LIN {X 0,Y 404.133,Z 307.643,A -85,B 0,C 180,E1 -10937.294,E2 -10937.294} C_VEL
LIN {X 0,Y 404.166,Z 307.632,A -85,B 0,C 180,E1 -10939.954,E2 -10939.954} C_VEL
LIN {X 0,Y 404.131,Z 307.643,A -85,B 0,C 180,E1 -10943.124,E2 -10943.124} C_VEL
LIN {X 0,Y 404.133,Z 307.632,A -85,B 0,C 180,E1 -10946.186,E2 -10946.186} C_VEL
LIN {X 0,Y 404.14,Z 307.645,A -85,B 0,C 180,E1 -10949.714,E2 -10949.714} C_VEL
LIN {X 0,Y 404.189,Z 307.62,A -85,B 0,C 180,E1 -10953.122,E2 -10953.122} C_VEL
LIN {X 0,Y 404.164,Z 307.633,A -85,B 0,C 180,E1 -10955.333,E2 -10955.333} C_VEL
LIN {X 0,Y 404.131,Z 307.638,A -85,B 0,C 180,E1 -10958.58,E2 -10958.58} C_VEL
LIN {X 0,Y 404.203,Z 307.615,A -85,B 0,C 180,E1 -10961.761,E2 -10961.761} C_VEL
LIN {X 0,Y 404.199,Z 307.63,A -85,B 0,C 180,E1 -10964.881,E2 -10964.881} C_VEL
LIN {X 0,Y 404.249,Z 307.619,A -85,B 0,C 180,E1 -10967.958,E2 -10967.958} C_VEL
LIN {X 0,Y 404.397,Z 307.598,A -85,B 0,C 180,E1 -10972.128,E2 -10972.128} C_VEL
LIN {X 0,Y 404.414,Z 307.606,A -85,B 0,C 180,E1 -10974.014,E2 -10974.014} C_VEL
LIN {X 0,Y 404.474,Z 307.59,A -85,B 0,C 180,E1 -10978.008,E2 -10978.008} C_VEL
LIN {X 0,Y 404.601,Z 307.557,A -85,B 0,C 180,E1 -10979.999,E2 -10979.999} C_VEL
LIN {X 0,Y 404.408,Z 307.602,A -85,B 0,C 180,E1 -10982.988,E2 -10982.988} C_VEL
LIN {X 0,Y 404.386,Z 307.608,A -85,B 0,C 180,E1 -10986.667,E2 -10986.667} C_VEL
LIN {X 0,Y 404.282,Z 307.606,A -85,B 0,C 180,E1 -10989.001,E2 -10989.001} C_VEL
LIN {X 0,Y 404.248,Z 307.619,A -85,B 0,C 180,E1 -10992.041,E2 -10992.041} C_VEL
LIN {X 0,Y 404.198,Z 307.637,A -85,B 0,C 180,E1 -10995.118,E2 -10995.118} C_VEL
LIN {X 0,Y 404.2,Z 307.621,A -85,B 0,C 180,E1 -10998.238,E2 -10998.238} C_VEL
LIN {X 0,Y 404.15,Z 307.639,A -85,B 0,C 180,E1 -11001.418,E2 -11001.418} C_VEL
LIN {X 0,Y 404.168,Z 307.641,A -85,B 0,C 180,E1 -11004.666,E2 -11004.666} C_VEL
LIN {X 0,Y 404.189,Z 307.62,A -85,B 0,C 180,E1 -11007.999,E2 -11007.999} C_VEL
LIN {X 0,Y 404.134,Z 307.642,A -85,B 0,C 180,E1 -11011.559,E2 -11011.559} C_VEL
LIN {X 0,Y 404.177,Z 307.629,A -85,B 0,C 180,E1 -11015.016,E2 -11015.016} C_VEL
LIN {X 0,Y 404.155,Z 307.641,A -85,B 0,C 180,E1 -11018.756,E2 -11018.756} C_VEL
LIN {X 0,Y 404.182,Z 307.631,A -85,B 0,C 180,E1 -11021.611,E2 -11021.611} C_VEL
LIN {X 0,Y 404.182,Z 307.636,A -85,B 0,C 180,E1 -11024.529,E2 -11024.529} C_VEL
LIN {X 0,Y 404.14,Z 307.611,A -85,B 0,C 180,E1 -11027.297,E2 -11027.297} C_VEL
LIN {X 0,Y 404.162,Z 307.627,A -85,B 0,C 180,E1 -11029.956,E2 -11029.956} C_VEL
LIN {X 0,Y 404.133,Z 307.64,A -85,B 0,C 180,E1 -11033.125,E2 -11033.125} C_VEL
LIN {X 0,Y 404.138,Z 307.624,A -85,B 0,C 180,E1 -11036.188,E2 -11036.188} C_VEL
LIN {X 0,Y 404.139,Z 307.637,A -85,B 0,C 180,E1 -11039.715,E2 -11039.715} C_VEL
LIN {X 0,Y 404.19,Z 307.638,A -85,B 0,C 180,E1 -11043.123,E2 -11043.123} C_VEL
LIN {X 0,Y 404.172,Z 307.64,A -85,B 0,C 180,E1 -11045.335,E2 -11045.335} C_VEL
LIN {X 0,Y 404.134,Z 307.647,A -85,B 0,C 180,E1 -11048.581,E2 -11048.581} C_VEL
LIN {X 0,Y 404.206,Z 307.638,A -85,B 0,C 180,E1 -11051.762,E2 -11051.762} C_VEL
LIN {X 0,Y 404.202,Z 307.637,A -85,B 0,C 180,E1 -11054.882,E2 -11054.882} C_VEL
LIN {X 0,Y 404.253,Z 307.632,A -85,B 0,C 180,E1 -11057.959,E2 -11057.959} C_VEL
LIN {X 0,Y 404.429,Z 307.611,A -85,B 0,C 180,E1 -11062.1,E2 -11062.1} C_VEL
LIN {X 0,Y 404.421,Z 307.611,A -85,B 0,C 180,E1 -11064.015,E2 -11064.015} C_VEL
LIN {X 0,Y 404.479,Z 307.603,A -85,B 0,C 180,E1 -11068.009,E2 -11068.009} C_VEL
LIN {X 0,Y 404.608,Z 307.588,A -85,B 0,C 180,E1 -11070,E2 -11070} C_VEL
LIN {X 0,Y 404.42,Z 307.611,A -85,B 0,C 180,E1 -11072.988,E2 -11072.988} C_VEL
LIN {X 0,Y 404.408,Z 307.613,A -85,B 0,C 180,E1 -11076.987,E2 -11076.987} C_VEL
LIN {X 0,Y 404.255,Z 307.632,A -85,B 0,C 180,E1 -11080.012,E2 -11080.012} C_VEL
LIN {X 0,Y 404.262,Z 307.63,A -85,B 0,C 180,E1 -11083.211,E2 -11083.211} C_VEL
LIN {X 0,Y 404.211,Z 307.636,A -85,B 0,C 180,E1 -11087.007,E2 -11087.007} C_VEL
LIN {X 0,Y 404.159,Z 307.643,A -85,B 0,C 180,E1 -11090.351,E2 -11090.351} C_VEL
LIN {X 0,Y 404.131,Z 307.644,A -85,B 0,C 180,E1 -11091.928,E2 -11091.928} C_VEL
LIN {X 0,Y 403.489,Z 307.726,A -85,B 0,C 180,E1 -11092.76,E2 -11092.76} C_VEL
LIN {X 0,Y 400.657,Z 308.081,A -85,B 0,C 180,E1 -11094.112,E2 -11094.112} C_VEL
LIN {X 0,Y 398.246,Z 308.382,A -85,B 0,C 180,E1 -11095.204,E2 -11095.204} C_VEL
LIN {X 0,Y 397.212,Z 308.509,A -85,B 0,C 180,E1 -11096.048,E2 -11096.048} C_VEL
LIN {X 0,Y 397.129,Z 308.517,A -85,B 0,C 180,E1 -11096.334,E2 -11096.334} C_VEL
LIN {X 0,Y 397.116,Z 308.508,A -85,B 0,C 180,E1 -11098.543,E2 -11098.543} C_VEL
LIN {X 0,Y 397.072,Z 308.523,A -85,B 0,C 180,E1 -11102.071,E2 -11102.071} C_VEL
LIN {X 0,Y 397.113,Z 308.499,A -85,B 0,C 180,E1 -11105.503,E2 -11105.503} C_VEL
LIN {X 0,Y 397.128,Z 308.517,A -85,B 0,C 180,E1 -11108.862,E2 -11108.862} C_VEL
LIN {X 0,Y 397.078,Z 308.487,A -85,B 0,C 180,E1 -11112.265,E2 -11112.265} C_VEL
LIN {X 0,Y 397.109,Z 308.511,A -85,B 0,C 180,E1 -11115.064,E2 -11115.064} C_VEL
LIN {X 0,Y 397.146,Z 308.508,A -85,B 0,C 180,E1 -11118.007,E2 -11118.007} C_VEL
LIN {X 0,Y 397.101,Z 308.521,A -85,B 0,C 180,E1 -11121.726,E2 -11121.726} C_VEL
LIN {X 0,Y 397.117,Z 308.506,A -85,B 0,C 180,E1 -11125.507,E2 -11125.507} C_VEL
LIN {X 0,Y 397.076,Z 308.527,A -85,B 0,C 180,E1 -11129.118,E2 -11129.118} C_VEL
LIN {X 0,Y 397.185,Z 308.492,A -85,B 0,C 180,E1 -11132.61,E2 -11132.61} C_VEL
LIN {X 0,Y 397.124,Z 308.515,A -85,B 0,C 180,E1 -11135.982,E2 -11135.982} C_VEL
LIN {X 0,Y 397.129,Z 308.499,A -85,B 0,C 180,E1 -11139.705,E2 -11139.705} C_VEL
LIN {X 0,Y 397.173,Z 308.501,A -85,B 0,C 180,E1 -11142.845,E2 -11142.845} C_VEL
LIN {X 0,Y 397.217,Z 308.506,A -85,B 0,C 180,E1 -11146.679,E2 -11146.679} C_VEL
LIN {X 0,Y 397.209,Z 308.478,A -85,B 0,C 180,E1 -11149.809,E2 -11149.809} C_VEL
LIN {X 0,Y 397.343,Z 308.485,A -85,B 0,C 180,E1 -11152.888,E2 -11152.888} C_VEL
LIN {X 0,Y 397.245,Z 308.504,A -85,B 0,C 180,E1 -11154.926,E2 -11154.926} C_VEL
LIN {X 0,Y 397.44,Z 308.465,A -85,B 0,C 180,E1 -11157.974,E2 -11157.974} C_VEL
LIN {X 0,Y 397.571,Z 308.432,A -85,B 0,C 180,E1 -11160.001,E2 -11160.001} C_VEL
LIN {X 0,Y 397.372,Z 308.486,A -85,B 0,C 180,E1 -11163.042,E2 -11163.042} C_VEL
LIN {X 0,Y 397.365,Z 308.484,A -85,B 0,C 180,E1 -11166.092,E2 -11166.092} C_VEL
LIN {X 0,Y 397.245,Z 308.474,A -85,B 0,C 180,E1 -11169.163,E2 -11169.163} C_VEL
LIN {X 0,Y 397.212,Z 308.497,A -85,B 0,C 180,E1 -11172.259,E2 -11172.259} C_VEL
LIN {X 0,Y 397.172,Z 308.504,A -85,B 0,C 180,E1 -11175.393,E2 -11175.393} C_VEL
LIN {X 0,Y 397.155,Z 308.491,A -85,B 0,C 180,E1 -11178.574,E2 -11178.574} C_VEL
LIN {X 0,Y 397.089,Z 308.516,A -85,B 0,C 180,E1 -11181.82,E2 -11181.82} C_VEL
LIN {X 0,Y 397.146,Z 308.502,A -85,B 0,C 180,E1 -11185.513,E2 -11185.513} C_VEL
LIN {X 0,Y 397.117,Z 308.511,A -85,B 0,C 180,E1 -11188.545,E2 -11188.545} C_VEL
LIN {X 0,Y 397.072,Z 308.523,A -85,B 0,C 180,E1 -11192.073,E2 -11192.073} C_VEL
LIN {X 0,Y 397.094,Z 308.513,A -85,B 0,C 180,E1 -11195.5,E2 -11195.5} C_VEL
LIN {X 0,Y 397.121,Z 308.51,A -85,B 0,C 180,E1 -11198.861,E2 -11198.861} C_VEL
LIN {X 0,Y 397.065,Z 308.528,A -85,B 0,C 180,E1 -11202.268,E2 -11202.268} C_VEL
LIN {X 0,Y 397.084,Z 308.518,A -85,B 0,C 180,E1 -11205.07,E2 -11205.07} C_VEL
LIN {X 0,Y 397.059,Z 308.516,A -85,B 0,C 180,E1 -11208.023,E2 -11208.023} C_VEL
LIN {X 0,Y 397.093,Z 308.521,A -85,B 0,C 180,E1 -11211.725,E2 -11211.725} C_VEL
LIN {X 0,Y 397.125,Z 308.515,A -85,B 0,C 180,E1 -11215.508,E2 -11215.508} C_VEL
LIN {X 0,Y 397.089,Z 308.524,A -85,B 0,C 180,E1 -11219.119,E2 -11219.119} C_VEL
LIN {X 0,Y 397.2,Z 308.757,A -85,B 0,C 180,E1 -11220.024,E2 -11220.024} C_VEL
LIN {X 0,Y 399.305,Z 319.657,A -85,B 0,C 180,E1 -11223.334,E2 -11223.334} C_VEL
LIN {X 0,Y 399.784,Z 324.864,A -85,B 0,C 180,E1 -11224.767,E2 -11224.767} C_VEL
LIN {X 0,Y 398.878,Z 336.233,A -85,B 0,C 180,E1 -11227.74,E2 -11227.74} C_VEL
LIN {X 0,Y 398.27,Z 344.064,A -85,B 0,C 180,E1 -11229.843,E2 -11229.843} C_VEL
LIN {X 0,Y 399.058,Z 348.58,A -85,B 0,C 180,E1 -11230.024,E2 -11230.024} C_VEL
LIN {X 0,Y 403.536,Z 373.485,A -85,B 0,C 180,E1 -11230.712,E2 -11230.712} C_VEL
LIN {X 0,Y 402.631,Z 449.002,A -85,B 0,C 180,E1 -11232.083,E2 -11232.083} C_VEL
LIN {X 0,Y 402.19,Z 459.766,A -85,B 0,C 180,E1 -11232.391,E2 -11232.391} C_VEL
LIN {X 0,Y 401.732,Z 468.864,A -85,B 0,C 180,E1 -11232.764,E2 -11232.764} C_VEL
LIN {X 0,Y 401.122,Z 479.226,A -85,B 0,C 180,E1 -11233.328,E2 -11233.328} C_VEL
LIN {X 0,Y 400.437,Z 488.358,A -85,B 0,C 180,E1 -11233.953,E2 -11233.953} C_VEL
LIN {X 0,Y 399.741,Z 497.354,A -85,B 0,C 180,E1 -11234.709,E2 -11234.709} C_VEL
LIN {X 0,Y 399.145,Z 504.953,A -85,B 0,C 180,E1 -11235.47,E2 -11235.47} C_VEL
LIN {X 0,Y 398.586,Z 511.877,A -85,B 0,C 180,E1 -11236.273,E2 -11236.273} C_VEL
LIN {X 0,Y 397.87,Z 520.701,A -85,B 0,C 180,E1 -11237.504,E2 -11237.504} C_VEL
LIN {X 0,Y 397.294,Z 526.901,A -85,B 0,C 180,E1 -11238.521,E2 -11238.521} C_VEL
LIN {X 0,Y 396.799,Z 533.44,A -85,B 0,C 180,E1 -11239.798,E2 -11239.798} C_VEL
LIN {X 0,Y 396.425,Z 537.941,A -85,B 0,C 180,E1 -11240.819,E2 -11240.819} C_VEL
LIN {X 0,Y 396.082,Z 543.432,A -85,B 0,C 180,E1 -11242.353,E2 -11242.353} C_VEL
LIN {X 0,Y 395.863,Z 547.756,A -85,B 0,C 180,E1 -11243.885,E2 -11243.885} C_VEL
LIN {X 0,Y 395.845,Z 550.124,A -85,B 0,C 180,E1 -11244.907,E2 -11244.907} C_VEL
LIN {X 0,Y 395.776,Z 551.921,A -85,B 0,C 180,E1 -11245.927,E2 -11245.927} C_VEL
LIN {X 0,Y 395.763,Z 554.365,A -85,B 0,C 180,E1 -11247.965,E2 -11247.965} C_VEL
LIN {X 0,Y 395.792,Z 554.955,A -85,B 0,C 180,E1 -11248.983,E2 -11248.983} C_VEL
LIN {X 0,Y 395.792,Z 554.955,A -85,B 0,C 180,E1 -11251.017,E2 -11251.017} C_VEL
LIN {X 0,Y 395.763,Z 554.365,A -85,B 0,C 180,E1 -11252.035,E2 -11252.035} C_VEL
LIN {X 0,Y 395.776,Z 551.921,A -85,B 0,C 180,E1 -11254.073,E2 -11254.073} C_VEL
LIN {X 0,Y 395.844,Z 550.124,A -85,B 0,C 180,E1 -11255.093,E2 -11255.093} C_VEL
LIN {X 0,Y 395.921,Z 546.518,A -85,B 0,C 180,E1 -11256.625,E2 -11256.625} C_VEL
LIN {X 0,Y 396.203,Z 541.773,A -85,B 0,C 180,E1 -11258.158,E2 -11258.158} C_VEL
LIN {X 0,Y 396.612,Z 535.751,A -85,B 0,C 180,E1 -11259.691,E2 -11259.691} C_VEL
LIN {X 0,Y 397.046,Z 529.653,A -85,B 0,C 180,E1 -11260.969,E2 -11260.969} C_VEL
LIN {X 0,Y 397.589,Z 523.954,A -85,B 0,C 180,E1 -11261.987,E2 -11261.987} C_VEL
LIN {X 0,Y 398.31,Z 515.4,A -85,B 0,C 180,E1 -11263.26,E2 -11263.26} C_VEL
LIN {X 0,Y 398.954,Z 507.218,A -85,B 0,C 180,E1 -11264.278,E2 -11264.278} C_VEL
LIN {X 0,Y 399.622,Z 498.841,A -85,B 0,C 180,E1 -11265.152,E2 -11265.152} C_VEL
LIN {X 0,Y 400.327,Z 489.99,A -85,B 0,C 180,E1 -11265.92,E2 -11265.92} C_VEL
LIN {X 0,Y 401.048,Z 480.233,A -85,B 0,C 180,E1 -11266.61,E2 -11266.61} C_VEL
LIN {X 0,Y 401.633,Z 470.151,A -85,B 0,C 180,E1 -11267.174,E2 -11267.174} C_VEL
LIN {X 0,Y 402.168,Z 460.641,A -85,B 0,C 180,E1 -11267.577,E2 -11267.577} C_VEL
LIN {X 0,Y 402.546,Z 450.332,A -85,B 0,C 180,E1 -11267.888,E2 -11267.888} C_VEL
LIN {X 0,Y 403.157,Z 408.947,A -85,B 0,C 180,E1 -11268.653,E2 -11268.653} C_VEL
LIN {X 0,Y 403.503,Z 373.005,A -85,B 0,C 180,E1 -11269.298,E2 -11269.298} C_VEL
LIN {X 0,Y 398.317,Z 344.544,A -85,B 0,C 180,E1 -11270.108,E2 -11270.108} C_VEL
LIN {X 0,Y 398.276,Z 343.513,A -85,B 0,C 180,E1 -11270.261,E2 -11270.261} C_VEL
LIN {X 0,Y 399.4,Z 330.246,A -85,B 0,C 180,E1 -11273.873,E2 -11273.873} C_VEL
LIN {X 0,Y 399.811,Z 323.063,A -85,B 0,C 180,E1 -11275.789,E2 -11275.789} C_VEL
LIN {X 0,Y 398.189,Z 313.707,A -85,B 0,C 180,E1 -11278.459,E2 -11278.459} C_VEL
LIN {X 0,Y 397.166,Z 308.6,A -85,B 0,C 180,E1 -11280.054,E2 -11280.054} C_VEL
LIN {X 0,Y 397.118,Z 308.518,A -85,B 0,C 180,E1 -11283.717,E2 -11283.717} C_VEL
LIN {X 0,Y 397.089,Z 308.519,A -85,B 0,C 180,E1 -11287.207,E2 -11287.207} C_VEL
LIN {X 0,Y 397.056,Z 308.506,A -85,B 0,C 180,E1 -11290.437,E2 -11290.437} C_VEL
LIN {X 0,Y 397.098,Z 308.523,A -85,B 0,C 180,E1 -11293.648,E2 -11293.648} C_VEL
LIN {X 0,Y 397.099,Z 308.518,A -85,B 0,C 180,E1 -11296.52,E2 -11296.52} C_VEL
LIN {X 0,Y 397.109,Z 308.512,A -85,B 0,C 180,E1 -11300.422,E2 -11300.422} C_VEL
LIN {X 0,Y 397.093,Z 308.519,A -85,B 0,C 180,E1 -11303.004,E2 -11303.004} C_VEL
LIN {X 0,Y 397.106,Z 308.507,A -85,B 0,C 180,E1 -11306.726,E2 -11306.726} C_VEL
LIN {X 0,Y 397.119,Z 308.514,A -85,B 0,C 180,E1 -11310.295,E2 -11310.295} C_VEL
LIN {X 0,Y 397.188,Z 308.492,A -85,B 0,C 180,E1 -11312.609,E2 -11312.609} C_VEL
LIN {X 0,Y 397.119,Z 308.516,A -85,B 0,C 180,E1 -11315.98,E2 -11315.98} C_VEL
LIN {X 0,Y 397.132,Z 308.502,A -85,B 0,C 180,E1 -11319.704,E2 -11319.704} C_VEL
LIN {X 0,Y 397.175,Z 308.493,A -85,B 0,C 180,E1 -11322.844,E2 -11322.844} C_VEL
LIN {X 0,Y 397.221,Z 308.501,A -85,B 0,C 180,E1 -11326.702,E2 -11326.702} C_VEL
LIN {X 0,Y 397.21,Z 308.48,A -85,B 0,C 180,E1 -11329.808,E2 -11329.808} C_VEL
LIN {X 0,Y 397.344,Z 308.479,A -85,B 0,C 180,E1 -11332.887,E2 -11332.887} C_VEL
LIN {X 0,Y 397.246,Z 308.501,A -85,B 0,C 180,E1 -11334.924,E2 -11334.924} C_VEL
LIN {X 0,Y 397.443,Z 308.466,A -85,B 0,C 180,E1 -11337.973,E2 -11337.973} C_VEL
LIN {X 0,Y 397.571,Z 308.432,A -85,B 0,C 180,E1 -11339.999,E2 -11339.999} C_VEL
LIN {X 0,Y 397.367,Z 308.479,A -85,B 0,C 180,E1 -11343.041,E2 -11343.041} C_VEL
LIN {X 0,Y 397.337,Z 308.484,A -85,B 0,C 180,E1 -11346.665,E2 -11346.665} C_VEL
LIN {X 0,Y 397.244,Z 308.479,A -85,B 0,C 180,E1 -11349.161,E2 -11349.161} C_VEL
LIN {X 0,Y 397.21,Z 308.496,A -85,B 0,C 180,E1 -11352.258,E2 -11352.258} C_VEL
LIN {X 0,Y 397.171,Z 308.51,A -85,B 0,C 180,E1 -11355.392,E2 -11355.392} C_VEL
LIN {X 0,Y 397.152,Z 308.496,A -85,B 0,C 180,E1 -11358.573,E2 -11358.573} C_VEL
LIN {X 0,Y 397.099,Z 308.515,A -85,B 0,C 180,E1 -11361.818,E2 -11361.818} C_VEL
LIN {X 0,Y 397.143,Z 308.506,A -85,B 0,C 180,E1 -11365.512,E2 -11365.512} C_VEL
LIN {X 0,Y 397.117,Z 308.504,A -85,B 0,C 180,E1 -11368.543,E2 -11368.543} C_VEL
LIN {X 0,Y 397.072,Z 308.522,A -85,B 0,C 180,E1 -11372.071,E2 -11372.071} C_VEL
LIN {X 0,Y 397.111,Z 308.511,A -85,B 0,C 180,E1 -11375.504,E2 -11375.504} C_VEL
LIN {X 0,Y 397.129,Z 308.515,A -85,B 0,C 180,E1 -11378.863,E2 -11378.863} C_VEL
LIN {X 0,Y 397.149,Z 308.51,A -85,B 0,C 180,E1 -11382.256,E2 -11382.256} C_VEL
LIN {X 0,Y 397.105,Z 308.511,A -85,B 0,C 180,E1 -11385.065,E2 -11385.065} C_VEL
LIN {X 0,Y 397.08,Z 308.486,A -85,B 0,C 180,E1 -11388.018,E2 -11388.018} C_VEL
LIN {X 0,Y 397.128,Z 308.517,A -85,B 0,C 180,E1 -11391.138,E2 -11391.138} C_VEL
LIN {X 0,Y 397.113,Z 308.499,A -85,B 0,C 180,E1 -11394.497,E2 -11394.497} C_VEL
LIN {X 0,Y 397.072,Z 308.523,A -85,B 0,C 180,E1 -11397.929,E2 -11397.929} C_VEL
LIN {X 0,Y 397.116,Z 308.508,A -85,B 0,C 180,E1 -11401.457,E2 -11401.457} C_VEL
LIN {X 0,Y 397.148,Z 308.517,A -85,B 0,C 180,E1 -11404.488,E2 -11404.488} C_VEL
LIN {X 0,Y 397.104,Z 308.521,A -85,B 0,C 180,E1 -11407.086,E2 -11407.086} C_VEL
LIN {X 0,Y 397.143,Z 308.518,A -85,B 0,C 180,E1 -11410.353,E2 -11410.353} C_VEL
LIN {X 0,Y 397.162,Z 308.514,A -85,B 0,C 180,E1 -11413.553,E2 -11413.553} C_VEL
LIN {X 0,Y 397.224,Z 308.508,A -85,B 0,C 180,E1 -11416.703,E2 -11416.703} C_VEL
LIN {X 0,Y 397.214,Z 308.509,A -85,B 0,C 180,E1 -11419.809,E2 -11419.809} C_VEL
LIN {X 0,Y 397.361,Z 308.491,A -85,B 0,C 180,E1 -11422.888,E2 -11422.888} C_VEL
LIN {X 0,Y 397.252,Z 308.504,A -85,B 0,C 180,E1 -11424.925,E2 -11424.925} C_VEL
LIN {X 0,Y 397.46,Z 308.77,A -85,B 0,C 180,E1 -11428.227,E2 -11428.227} C_VEL
LIN {X 0,Y 397.65,Z 308.874,A -85,B 0,C 180,E1 -11430,E2 -11430} C_VEL
LIN {X 0,Y 397.378,Z 308.565,A -85,B 0,C 180,E1 -11433.041,E2 -11433.041} C_VEL
LIN {X 0,Y 397.361,Z 308.491,A -85,B 0,C 180,E1 -11437.112,E2 -11437.112} C_VEL
LIN {X 0,Y 397.214,Z 308.509,A -85,B 0,C 180,E1 -11440.191,E2 -11440.191} C_VEL
LIN {X 0,Y 397.222,Z 308.508,A -85,B 0,C 180,E1 -11443.321,E2 -11443.321} C_VEL
LIN {X 0,Y 397.177,Z 308.513,A -85,B 0,C 180,E1 -11447.155,E2 -11447.155} C_VEL
LIN {X 0,Y 397.098,Z 308.522,A -85,B 0,C 180,E1 -11450.73,E2 -11450.73} C_VEL
LIN {X 0,Y 397.128,Z 308.519,A -85,B 0,C 180,E1 -11454.018,E2 -11454.018} C_VEL
LIN {X 0,Y 397.129,Z 308.517,A -85,B 0,C 180,E1 -11456.334,E2 -11456.334} C_VEL
LIN {X 0,Y 396.459,Z 308.602,A -85,B 0,C 180,E1 -11457.181,E2 -11457.181} C_VEL
LIN {X 0,Y 393.584,Z 308.949,A -85,B 0,C 180,E1 -11458.556,E2 -11458.556} C_VEL
LIN {X 0,Y 391.145,Z 309.251,A -85,B 0,C 180,E1 -11459.668,E2 -11459.668} C_VEL
LIN {X 0,Y 390.093,Z 309.389,A -85,B 0,C 180,E1 -11460.528,E2 -11460.528} C_VEL
LIN {X 0,Y 390.005,Z 309.398,A -85,B 0,C 180,E1 -11460.819,E2 -11460.819} C_VEL
LIN {X 0,Y 390.062,Z 309.374,A -85,B 0,C 180,E1 -11464.024,E2 -11464.024} C_VEL
LIN {X 0,Y 390.039,Z 309.402,A -85,B 0,C 180,E1 -11467.551,E2 -11467.551} C_VEL
LIN {X 0,Y 390.069,Z 309.369,A -85,B 0,C 180,E1 -11470.824,E2 -11470.824} C_VEL
LIN {X 0,Y 390.056,Z 309.387,A -85,B 0,C 180,E1 -11474.643,E2 -11474.643} C_VEL
LIN {X 0,Y 390.111,Z 309.387,A -85,B 0,C 180,E1 -11477.613,E2 -11477.613} C_VEL
LIN {X 0,Y 390.087,Z 309.389,A -85,B 0,C 180,E1 -11480.908,E2 -11480.908} C_VEL
LIN {X 0,Y 390.077,Z 309.385,A -85,B 0,C 180,E1 -11484.793,E2 -11484.793} C_VEL
LIN {X 0,Y 390.019,Z 309.401,A -85,B 0,C 180,E1 -11488.496,E2 -11488.496} C_VEL
LIN {X 0,Y 390.108,Z 309.373,A -85,B 0,C 180,E1 -11492.07,E2 -11492.07} C_VEL
LIN {X 0,Y 390.071,Z 309.396,A -85,B 0,C 180,E1 -11495.519,E2 -11495.519} C_VEL
LIN {X 0,Y 390.053,Z 309.389,A -85,B 0,C 180,E1 -11498.878,E2 -11498.878} C_VEL
LIN {X 0,Y 390.119,Z 309.374,A -85,B 0,C 180,E1 -11502.167,E2 -11502.167} C_VEL
LIN {X 0,Y 390.138,Z 309.387,A -85,B 0,C 180,E1 -11505.393,E2 -11505.393} C_VEL
LIN {X 0,Y 390.14,Z 309.371,A -85,B 0,C 180,E1 -11508.572,E2 -11508.572} C_VEL
LIN {X 0,Y 390.299,Z 309.355,A -85,B 0,C 180,E1 -11512.032,E2 -11512.032} C_VEL
LIN {X 0,Y 390.217,Z 309.381,A -85,B 0,C 180,E1 -11514.834,E2 -11514.834} C_VEL
LIN {X 0,Y 390.409,Z 309.34,A -85,B 0,C 180,E1 -11517.937,E2 -11517.937} C_VEL
LIN {X 0,Y 390.54,Z 309.307,A -85,B 0,C 180,E1 -11520.001,E2 -11520.001} C_VEL
LIN {X 0,Y 390.306,Z 309.366,A -85,B 0,C 180,E1 -11523.097,E2 -11523.097} C_VEL
LIN {X 0,Y 390.318,Z 309.363,A -85,B 0,C 180,E1 -11526.203,E2 -11526.203} C_VEL
LIN {X 0,Y 390.197,Z 309.351,A -85,B 0,C 180,E1 -11529.33,E2 -11529.33} C_VEL
LIN {X 0,Y 390.187,Z 309.377,A -85,B 0,C 180,E1 -11533.439,E2 -11533.439} C_VEL
